   1:  PR[GP1:91,1] = PR[GP1:90,1] + -14.975;
   1:  PR[GP1:91,2] = PR[GP1:90,2] + 38.981;
   1:L PR[91] R[100]mm/sec CNT100;
   1:  PR[GP1:91,1] = PR[GP1:90,1] + -26.046;
   1:  PR[GP1:91,2] = PR[GP1:90,2] + 38.779;
   1:L PR[91] R[100]mm/sec CNT100;
   1:  PR[GP1:91,1] = PR[GP1:90,1] + -28.313;
   1:  PR[GP1:91,2] = PR[GP1:90,2] + 38.036;
   1:L PR[91] R[100]mm/sec CNT100;
   1:  PR[GP1:91,1] = PR[GP1:90,1] + -39.636;
   1:  PR[GP1:91,2] = PR[GP1:90,2] + 33.857;
   1:L PR[91] R[100]mm/sec CNT100;
   1:  PR[GP1:91,1] = PR[GP1:90,1] + -40.541;
   1:  PR[GP1:91,2] = PR[GP1:90,2] + 33.140;
   1:L PR[91] R[100]mm/sec CNT100;
   1:  PR[GP1:91,1] = PR[GP1:90,1] + -50.506;
   1:  PR[GP1:91,2] = PR[GP1:90,2] + 24.916;
   1:L PR[91] R[100]mm/sec CNT100;
   1:  PR[GP1:91,1] = PR[GP1:90,1] + -52.333;
   1:  PR[GP1:91,2] = PR[GP1:90,2] + 21.827;
   1:L PR[91] R[100]mm/sec CNT100;
   1:  PR[GP1:91,1] = PR[GP1:90,1] + -57.539;
   1:  PR[GP1:91,2] = PR[GP1:90,2] + 13.132;
   1:L PR[91] R[100]mm/sec CNT100;
   1:  PR[GP1:91,1] = PR[GP1:90,1] + -57.566;
   1:  PR[GP1:91,2] = PR[GP1:90,2] + 13.038;
   1:L PR[91] R[100]mm/sec CNT100;
   1:  PR[GP1:91,1] = PR[GP1:90,1] + -57.585;
   1:  PR[GP1:91,2] = PR[GP1:90,2] + 12.836;
   1:L PR[91] R[100]mm/sec CNT100;
   1:  PR[GP1:91,1] = PR[GP1:90,1] + -59.969;
   1:  PR[GP1:91,2] = PR[GP1:90,2] + -0.100;
   1:L PR[91] R[100]mm/sec CNT100;
   1:  PR[GP1:91,1] = PR[GP1:90,1] + -59.943;
   1:  PR[GP1:91,2] = PR[GP1:90,2] + -0.390;
   1:L PR[91] R[100]mm/sec CNT100;
   1:  PR[GP1:91,1] = PR[GP1:90,1] + -57.573;
   1:  PR[GP1:91,2] = PR[GP1:90,2] + -13.159;
   1:L PR[91] R[100]mm/sec CNT100;
   1:  PR[GP1:91,1] = PR[GP1:90,1] + -57.531;
   1:  PR[GP1:91,2] = PR[GP1:90,2] + -13.299;
   1:L PR[91] R[100]mm/sec CNT100;
   1:  PR[GP1:91,1] = PR[GP1:90,1] + -57.460;
   1:  PR[GP1:91,2] = PR[GP1:90,2] + -13.440;
   1:L PR[91] R[100]mm/sec CNT100;
   1:  PR[GP1:91,1] = PR[GP1:90,1] + -52.333;
   1:  PR[GP1:91,2] = PR[GP1:90,2] + -21.969;
   1:L PR[91] R[100]mm/sec CNT100;
   1:  PR[GP1:91,1] = PR[GP1:90,1] + -50.500;
   1:  PR[GP1:91,2] = PR[GP1:90,2] + -25.067;
   1:L PR[91] R[100]mm/sec CNT100;
   1:  PR[GP1:91,1] = PR[GP1:90,1] + -40.531;
   1:  PR[GP1:91,2] = PR[GP1:90,2] + -33.290;
   1:L PR[91] R[100]mm/sec CNT100;
   1:  PR[GP1:91,1] = PR[GP1:90,1] + -39.625;
   1:  PR[GP1:91,2] = PR[GP1:90,2] + -34.007;
   1:L PR[91] R[100]mm/sec CNT100;
   1:  PR[GP1:91,1] = PR[GP1:90,1] + -28.299;
   1:  PR[GP1:91,2] = PR[GP1:90,2] + -38.182;
   1:L PR[91] R[100]mm/sec CNT100;
   1:  PR[GP1:91,1] = PR[GP1:90,1] + -26.031;
   1:  PR[GP1:91,2] = PR[GP1:90,2] + -38.926;
   1:L PR[91] R[100]mm/sec CNT100;
   1:  PR[GP1:91,1] = PR[GP1:90,1] + -14.960;
   1:  PR[GP1:91,2] = PR[GP1:90,2] + -39.122;
   1:L PR[91] R[100]mm/sec CNT100;
   1:  PR[GP1:91,1] = PR[GP1:90,1] + -11.340;
   1:  PR[GP1:91,2] = PR[GP1:90,2] + -38.993;
   1:L PR[91] R[100]mm/sec CNT100;
   1:  PR[GP1:91,1] = PR[GP1:90,1] + -1.863;
   1:  PR[GP1:91,2] = PR[GP1:90,2] + -36.043;
   1:L PR[91] R[100]mm/sec CNT100;
   1:  PR[GP1:91,1] = PR[GP1:90,1] + 2.073;
   1:  PR[GP1:91,2] = PR[GP1:90,2] + -36.042;
   1:L PR[91] R[100]mm/sec CNT100;
   1:  PR[GP1:91,1] = PR[GP1:90,1] + 11.551;
   1:  PR[GP1:91,2] = PR[GP1:90,2] + -38.993;
   1:L PR[91] R[100]mm/sec CNT100;
   1:  PR[GP1:91,1] = PR[GP1:90,1] + 15.171;
   1:  PR[GP1:91,2] = PR[GP1:90,2] + -39.122;
   1:L PR[91] R[100]mm/sec CNT100;
   1:  PR[GP1:91,1] = PR[GP1:90,1] + 26.243;
   1:  PR[GP1:91,2] = PR[GP1:90,2] + -38.926;
   1:L PR[91] R[100]mm/sec CNT100;
   1:  PR[GP1:91,1] = PR[GP1:90,1] + 28.510;
   1:  PR[GP1:91,2] = PR[GP1:90,2] + -38.182;
   1:L PR[91] R[100]mm/sec CNT100;
   1:  PR[GP1:91,1] = PR[GP1:90,1] + 39.837;
   1:  PR[GP1:91,2] = PR[GP1:90,2] + -34.010;
   1:L PR[91] R[100]mm/sec CNT100;
   1:  PR[GP1:91,1] = PR[GP1:90,1] + 40.743;
   1:  PR[GP1:91,2] = PR[GP1:90,2] + -33.293;
   1:L PR[91] R[100]mm/sec CNT100;
   1:  PR[GP1:91,1] = PR[GP1:90,1] + 50.715;
   1:  PR[GP1:91,2] = PR[GP1:90,2] + -25.059;
   1:L PR[91] R[100]mm/sec CNT100;
   1:  PR[GP1:91,1] = PR[GP1:90,1] + 50.759;
   1:  PR[GP1:91,2] = PR[GP1:90,2] + -24.985;
   1:L PR[91] R[100]mm/sec CNT100;
   1:  PR[GP1:91,1] = PR[GP1:90,1] + 52.546;
   1:  PR[GP1:91,2] = PR[GP1:90,2] + -21.970;
   1:L PR[91] R[100]mm/sec CNT100;
   1:  PR[GP1:91,1] = PR[GP1:90,1] + 57.750;
   1:  PR[GP1:91,2] = PR[GP1:90,2] + -13.299;
   1:L PR[91] R[100]mm/sec CNT100;
   1:  PR[GP1:91,1] = PR[GP1:90,1] + 57.777;
   1:  PR[GP1:91,2] = PR[GP1:90,2] + -13.208;
   1:L PR[91] R[100]mm/sec CNT100;
   1:  PR[GP1:91,1] = PR[GP1:90,1] + 57.796;
   1:  PR[GP1:91,2] = PR[GP1:90,2] + -13.001;
   1:L PR[91] R[100]mm/sec CNT100;
   1:  PR[GP1:91,1] = PR[GP1:90,1] + 60.182;
   1:  PR[GP1:91,2] = PR[GP1:90,2] + -0.045;
   1:L PR[91] R[100]mm/sec CNT100;
   1:  PR[GP1:91,1] = PR[GP1:90,1] + 60.155;
   1:  PR[GP1:91,2] = PR[GP1:90,2] + 0.256;
   1:L PR[91] R[100]mm/sec CNT100;
   1:  PR[GP1:91,1] = PR[GP1:90,1] + 57.786;
   1:  PR[GP1:91,2] = PR[GP1:90,2] + 13.034;
   1:L PR[91] R[100]mm/sec CNT100;
   1:  PR[GP1:91,1] = PR[GP1:90,1] + 57.746;
   1:  PR[GP1:91,2] = PR[GP1:90,2] + 13.170;
   1:L PR[91] R[100]mm/sec CNT100;
   1:  PR[GP1:91,1] = PR[GP1:90,1] + 57.674;
   1:  PR[GP1:91,2] = PR[GP1:90,2] + 13.309;
   1:L PR[91] R[100]mm/sec CNT100;
   1:  PR[GP1:91,1] = PR[GP1:90,1] + 52.546;
   1:  PR[GP1:91,2] = PR[GP1:90,2] + 21.827;
   1:L PR[91] R[100]mm/sec CNT100;
   1:  PR[GP1:91,1] = PR[GP1:90,1] + 50.718;
   1:  PR[GP1:91,2] = PR[GP1:90,2] + 24.910;
   1:L PR[91] R[100]mm/sec CNT100;
   1:  PR[GP1:91,1] = PR[GP1:90,1] + 40.752;
   1:  PR[GP1:91,2] = PR[GP1:90,2] + 33.144;
   1:L PR[91] R[100]mm/sec CNT100;
   1:  PR[GP1:91,1] = PR[GP1:90,1] + 39.848;
   1:  PR[GP1:91,2] = PR[GP1:90,2] + 33.860;
   1:L PR[91] R[100]mm/sec CNT100;
   1:  PR[GP1:91,1] = PR[GP1:90,1] + 28.524;
   1:  PR[GP1:91,2] = PR[GP1:90,2] + 38.036;
   1:L PR[91] R[100]mm/sec CNT100;
   1:  PR[GP1:91,1] = PR[GP1:90,1] + 26.257;
   1:  PR[GP1:91,2] = PR[GP1:90,2] + 38.780;
   1:L PR[91] R[100]mm/sec CNT100;
   1:  PR[GP1:91,1] = PR[GP1:90,1] + 15.186;
   1:  PR[GP1:91,2] = PR[GP1:90,2] + 38.980;
   1:L PR[91] R[100]mm/sec CNT100;
   1:  PR[GP1:91,1] = PR[GP1:90,1] + 11.565;
   1:  PR[GP1:91,2] = PR[GP1:90,2] + 38.851;
   1:L PR[91] R[100]mm/sec CNT100;
   1:  PR[GP1:91,1] = PR[GP1:90,1] + 2.071;
   1:  PR[GP1:91,2] = PR[GP1:90,2] + 35.917;
   1:L PR[91] R[100]mm/sec CNT100;
   1:  ! -- Layer/Ebene 129 -- !;
   1:  PR[91] = PR[90];
   1:  PR[GP1:91,1] = PR[GP1:90,1] + -1.835;
   1:  PR[GP1:91,2] = PR[GP1:90,2] + 36.091;
   1:  PR[GP1:91,3] = PR[GP1:90,3] + 78.995;
   1:L PR[91] R[100]mm/sec CNT100;
   1:  PR[GP1:91,1] = PR[GP1:90,1] + -11.057;
   1:  PR[GP1:91,2] = PR[GP1:90,2] + 38.940;
   1:L PR[91] R[100]mm/sec CNT100;
   1:  PR[GP1:91,1] = PR[GP1:90,1] + -15.013;
   1:  PR[GP1:91,2] = PR[GP1:90,2] + 39.082;
   1:L PR[91] R[100]mm/sec CNT100;
   1:  PR[GP1:91,1] = PR[GP1:90,1] + -25.784;
   1:  PR[GP1:91,2] = PR[GP1:90,2] + 38.885;
   1:L PR[91] R[100]mm/sec CNT100;
   1:  PR[GP1:91,1] = PR[GP1:90,1] + -28.381;
   1:  PR[GP1:91,2] = PR[GP1:90,2] + 38.034;
   1:L PR[91] R[100]mm/sec CNT100;
   1:  PR[GP1:91,1] = PR[GP1:90,1] + -39.414;
   1:  PR[GP1:91,2] = PR[GP1:90,2] + 33.962;
   1:L PR[91] R[100]mm/sec CNT100;
   1:  PR[GP1:91,1] = PR[GP1:90,1] + -40.601;
   1:  PR[GP1:91,2] = PR[GP1:90,2] + 33.023;
   1:L PR[91] R[100]mm/sec CNT100;
   1:  PR[GP1:91,1] = PR[GP1:90,1] + -50.321;
   1:  PR[GP1:91,2] = PR[GP1:90,2] + 25.000;
   1:L PR[91] R[100]mm/sec CNT100;
   1:  PR[GP1:91,1] = PR[GP1:90,1] + -55.806;
   1:  PR[GP1:91,2] = PR[GP1:90,2] + 15.729;
   1:L PR[91] R[100]mm/sec CNT100;
   1:  PR[GP1:91,1] = PR[GP1:90,1] + -57.336;
   1:  PR[GP1:91,2] = PR[GP1:90,2] + 13.173;
   1:L PR[91] R[100]mm/sec CNT100;
   1:  PR[GP1:91,1] = PR[GP1:90,1] + -57.342;
   1:  PR[GP1:91,2] = PR[GP1:90,2] + 13.142;
   1:L PR[91] R[100]mm/sec CNT100;
   1:  PR[GP1:91,1] = PR[GP1:90,1] + -59.783;
   1:  PR[GP1:91,2] = PR[GP1:90,2] + -0.100;
   1:L PR[91] R[100]mm/sec CNT100;
   1:  PR[GP1:91,1] = PR[GP1:90,1] + -59.771;
   1:  PR[GP1:91,2] = PR[GP1:90,2] + -0.233;
   1:L PR[91] R[100]mm/sec CNT100;
   1:  PR[GP1:91,1] = PR[GP1:90,1] + -57.334;
   1:  PR[GP1:91,2] = PR[GP1:90,2] + -13.322;
   1:L PR[91] R[100]mm/sec CNT100;
   1:  PR[GP1:91,1] = PR[GP1:90,1] + -55.806;
   1:  PR[GP1:91,2] = PR[GP1:90,2] + -15.873;
   1:L PR[91] R[100]mm/sec CNT100;
   1:  PR[GP1:91,1] = PR[GP1:90,1] + -50.315;
   1:  PR[GP1:91,2] = PR[GP1:90,2] + -25.151;
   1:L PR[91] R[100]mm/sec CNT100;
   1:  PR[GP1:91,1] = PR[GP1:90,1] + -40.591;
   1:  PR[GP1:91,2] = PR[GP1:90,2] + -33.172;
   1:L PR[91] R[100]mm/sec CNT100;
   1:  PR[GP1:91,1] = PR[GP1:90,1] + -39.404;
   1:  PR[GP1:91,2] = PR[GP1:90,2] + -34.112;
   1:L PR[91] R[100]mm/sec CNT100;
   1:  PR[GP1:91,1] = PR[GP1:90,1] + -28.368;
   1:  PR[GP1:91,2] = PR[GP1:90,2] + -38.180;
   1:L PR[91] R[100]mm/sec CNT100;
   1:  PR[GP1:91,1] = PR[GP1:90,1] + -25.770;
   1:  PR[GP1:91,2] = PR[GP1:90,2] + -39.032;
   1:L PR[91] R[100]mm/sec CNT100;
   1:  PR[GP1:91,1] = PR[GP1:90,1] + -14.999;
   1:  PR[GP1:91,2] = PR[GP1:90,2] + -39.223;
   1:L PR[91] R[100]mm/sec CNT100;
   1:  PR[GP1:91,1] = PR[GP1:90,1] + -11.043;
   1:  PR[GP1:91,2] = PR[GP1:90,2] + -39.082;
   1:L PR[91] R[100]mm/sec CNT100;
   1:  PR[GP1:91,1] = PR[GP1:90,1] + -1.838;
   1:  PR[GP1:91,2] = PR[GP1:90,2] + -36.217;
   1:L PR[91] R[100]mm/sec CNT100;
   1:  PR[GP1:91,1] = PR[GP1:90,1] + 2.048;
   1:  PR[GP1:91,2] = PR[GP1:90,2] + -36.216;
   1:L PR[91] R[100]mm/sec CNT100;
   1:  PR[GP1:91,1] = PR[GP1:90,1] + 11.254;
   1:  PR[GP1:91,2] = PR[GP1:90,2] + -39.081;
   1:L PR[91] R[100]mm/sec CNT100;
   1:  PR[GP1:91,1] = PR[GP1:90,1] + 15.210;
   1:  PR[GP1:91,2] = PR[GP1:90,2] + -39.222;
   1:L PR[91] R[100]mm/sec CNT100;
   1:  PR[GP1:91,1] = PR[GP1:90,1] + 25.982;
   1:  PR[GP1:91,2] = PR[GP1:90,2] + -39.032;
   1:L PR[91] R[100]mm/sec CNT100;
   1:  PR[GP1:91,1] = PR[GP1:90,1] + 28.579;
   1:  PR[GP1:91,2] = PR[GP1:90,2] + -38.180;
   1:L PR[91] R[100]mm/sec CNT100;
   1:  PR[GP1:91,1] = PR[GP1:90,1] + 39.616;
   1:  PR[GP1:91,2] = PR[GP1:90,2] + -34.115;
   1:L PR[91] R[100]mm/sec CNT100;
   1:  PR[GP1:91,1] = PR[GP1:90,1] + 40.803;
   1:  PR[GP1:91,2] = PR[GP1:90,2] + -33.175;
   1:L PR[91] R[100]mm/sec CNT100;
   1:  PR[GP1:91,1] = PR[GP1:90,1] + 50.530;
   1:  PR[GP1:91,2] = PR[GP1:90,2] + -25.143;
   1:L PR[91] R[100]mm/sec CNT100;
   1:  PR[GP1:91,1] = PR[GP1:90,1] + 50.766;
   1:  PR[GP1:91,2] = PR[GP1:90,2] + -24.753;
   1:L PR[91] R[100]mm/sec CNT100;
   1:  PR[GP1:91,1] = PR[GP1:90,1] + 56.019;
   1:  PR[GP1:91,2] = PR[GP1:90,2] + -15.886;
   1:L PR[91] R[100]mm/sec CNT100;
   1:  PR[GP1:91,1] = PR[GP1:90,1] + 57.546;
   1:  PR[GP1:91,2] = PR[GP1:90,2] + -13.341;
   1:L PR[91] R[100]mm/sec CNT100;
   1:  PR[GP1:91,1] = PR[GP1:90,1] + 59.996;
   1:  PR[GP1:91,2] = PR[GP1:90,2] + -0.045;
   1:L PR[91] R[100]mm/sec CNT100;
   1:  PR[GP1:91,1] = PR[GP1:90,1] + 59.983;
   1:  PR[GP1:91,2] = PR[GP1:90,2] + 0.095;
   1:L PR[91] R[100]mm/sec CNT100;
   1:  PR[GP1:91,1] = PR[GP1:90,1] + 57.548;
   1:  PR[GP1:91,2] = PR[GP1:90,2] + 13.193;
   1:L PR[91] R[100]mm/sec CNT100;
   1:  PR[GP1:91,1] = PR[GP1:90,1] + 56.019;
   1:  PR[GP1:91,2] = PR[GP1:90,2] + 15.742;
   1:L PR[91] R[100]mm/sec CNT100;
   1:  PR[GP1:91,1] = PR[GP1:90,1] + 50.533;
   1:  PR[GP1:91,2] = PR[GP1:90,2] + 24.994;
   1:L PR[91] R[100]mm/sec CNT100;
   1:  PR[GP1:91,1] = PR[GP1:90,1] + 40.812;
   1:  PR[GP1:91,2] = PR[GP1:90,2] + 33.026;
   1:L PR[91] R[100]mm/sec CNT100;
   1:  PR[GP1:91,1] = PR[GP1:90,1] + 39.626;
   1:  PR[GP1:91,2] = PR[GP1:90,2] + 33.965;
   1:L PR[91] R[100]mm/sec CNT100;
   1:  PR[GP1:91,1] = PR[GP1:90,1] + 28.592;
   1:  PR[GP1:91,2] = PR[GP1:90,2] + 38.034;
   1:L PR[91] R[100]mm/sec CNT100;
   1:  PR[GP1:91,1] = PR[GP1:90,1] + 25.995;
   1:  PR[GP1:91,2] = PR[GP1:90,2] + 38.886;
   1:L PR[91] R[100]mm/sec CNT100;
   1:  PR[GP1:91,1] = PR[GP1:90,1] + 15.224;
   1:  PR[GP1:91,2] = PR[GP1:90,2] + 39.081;
   1:L PR[91] R[100]mm/sec CNT100;
   1:  PR[GP1:91,1] = PR[GP1:90,1] + 11.268;
   1:  PR[GP1:91,2] = PR[GP1:90,2] + 38.939;
   1:L PR[91] R[100]mm/sec CNT100;
   1:  PR[GP1:91,1] = PR[GP1:90,1] + 2.046;
   1:  PR[GP1:91,2] = PR[GP1:90,2] + 36.090;
   1:L PR[91] R[100]mm/sec CNT100;
   1:  ! -- Layer/Ebene 130 -- !;
   1:  PR[91] = PR[90];
   1:  PR[GP1:91,1] = PR[GP1:90,1] + -1.810;
   1:  PR[GP1:91,2] = PR[GP1:90,2] + 36.264;
   1:  PR[GP1:91,3] = PR[GP1:90,3] + 79.605;
   1:L PR[91] R[100]mm/sec CNT100;
   1:  PR[GP1:91,1] = PR[GP1:90,1] + -10.759;
   1:  PR[GP1:91,2] = PR[GP1:90,2] + 39.029;
   1:L PR[91] R[100]mm/sec CNT100;
   1:  PR[GP1:91,1] = PR[GP1:90,1] + -15.051;
   1:  PR[GP1:91,2] = PR[GP1:90,2] + 39.183;
   1:L PR[91] R[100]mm/sec CNT100;
   1:  PR[GP1:91,1] = PR[GP1:90,1] + -25.523;
   1:  PR[GP1:91,2] = PR[GP1:90,2] + 38.991;
   1:L PR[91] R[100]mm/sec CNT100;
   1:  PR[GP1:91,1] = PR[GP1:90,1] + -28.449;
   1:  PR[GP1:91,2] = PR[GP1:90,2] + 38.032;
   1:L PR[91] R[100]mm/sec CNT100;
   1:  PR[GP1:91,1] = PR[GP1:90,1] + -39.193;
   1:  PR[GP1:91,2] = PR[GP1:90,2] + 34.067;
   1:L PR[91] R[100]mm/sec CNT100;
   1:  PR[GP1:91,1] = PR[GP1:90,1] + -40.661;
   1:  PR[GP1:91,2] = PR[GP1:90,2] + 32.905;
   1:L PR[91] R[100]mm/sec CNT100;
   1:  PR[GP1:91,1] = PR[GP1:90,1] + -50.136;
   1:  PR[GP1:91,2] = PR[GP1:90,2] + 25.084;
   1:L PR[91] R[100]mm/sec CNT100;
   1:  PR[GP1:91,1] = PR[GP1:90,1] + -57.164;
   1:  PR[GP1:91,2] = PR[GP1:90,2] + 13.211;
   1:L PR[91] R[100]mm/sec CNT100;
   1:  PR[GP1:91,1] = PR[GP1:90,1] + -58.384;
   1:  PR[GP1:91,2] = PR[GP1:90,2] + 6.480;
   1:L PR[91] R[100]mm/sec CNT100;
   1:  PR[GP1:91,1] = PR[GP1:90,1] + -59.592;
   1:  PR[GP1:91,2] = PR[GP1:90,2] + -0.072;
   1:L PR[91] R[100]mm/sec CNT100;
   1:  PR[GP1:91,1] = PR[GP1:90,1] + -58.384;
   1:  PR[GP1:91,2] = PR[GP1:90,2] + -6.623;
   1:L PR[91] R[100]mm/sec CNT100;
   1:  PR[GP1:91,1] = PR[GP1:90,1] + -57.162;
   1:  PR[GP1:91,2] = PR[GP1:90,2] + -13.359;
   1:L PR[91] R[100]mm/sec CNT100;
   1:  PR[GP1:91,1] = PR[GP1:90,1] + -50.131;
   1:  PR[GP1:91,2] = PR[GP1:90,2] + -25.235;
   1:L PR[91] R[100]mm/sec CNT100;
   1:  PR[GP1:91,1] = PR[GP1:90,1] + -40.651;
   1:  PR[GP1:91,2] = PR[GP1:90,2] + -33.054;
   1:L PR[91] R[100]mm/sec CNT100;
   1:  PR[GP1:91,1] = PR[GP1:90,1] + -39.183;
   1:  PR[GP1:91,2] = PR[GP1:90,2] + -34.216;
   1:L PR[91] R[100]mm/sec CNT100;
   1:  PR[GP1:91,1] = PR[GP1:90,1] + -28.437;
   1:  PR[GP1:91,2] = PR[GP1:90,2] + -38.178;
   1:L PR[91] R[100]mm/sec CNT100;
   1:  PR[GP1:91,1] = PR[GP1:90,1] + -25.509;
   1:  PR[GP1:91,2] = PR[GP1:90,2] + -39.138;
   1:L PR[91] R[100]mm/sec CNT100;
   1:  PR[GP1:91,1] = PR[GP1:90,1] + -15.037;
   1:  PR[GP1:91,2] = PR[GP1:90,2] + -39.324;
   1:L PR[91] R[100]mm/sec CNT100;
   1:  PR[GP1:91,1] = PR[GP1:90,1] + -10.746;
   1:  PR[GP1:91,2] = PR[GP1:90,2] + -39.171;
   1:L PR[91] R[100]mm/sec CNT100;
   1:  PR[GP1:91,1] = PR[GP1:90,1] + -1.812;
   1:  PR[GP1:91,2] = PR[GP1:90,2] + -36.391;
   1:L PR[91] R[100]mm/sec CNT100;
   1:  PR[GP1:91,1] = PR[GP1:90,1] + 2.023;
   1:  PR[GP1:91,2] = PR[GP1:90,2] + -36.389;
   1:L PR[91] R[100]mm/sec CNT100;
   1:  PR[GP1:91,1] = PR[GP1:90,1] + 10.958;
   1:  PR[GP1:91,2] = PR[GP1:90,2] + -39.170;
   1:L PR[91] R[100]mm/sec CNT100;
   1:  PR[GP1:91,1] = PR[GP1:90,1] + 15.249;
   1:  PR[GP1:91,2] = PR[GP1:90,2] + -39.323;
   1:L PR[91] R[100]mm/sec CNT100;
   1:  PR[GP1:91,1] = PR[GP1:90,1] + 25.721;
   1:  PR[GP1:91,2] = PR[GP1:90,2] + -39.138;
   1:L PR[91] R[100]mm/sec CNT100;
   1:  PR[GP1:91,1] = PR[GP1:90,1] + 28.648;
   1:  PR[GP1:91,2] = PR[GP1:90,2] + -38.178;
   1:L PR[91] R[100]mm/sec CNT100;
   1:  PR[GP1:91,1] = PR[GP1:90,1] + 39.395;
   1:  PR[GP1:91,2] = PR[GP1:90,2] + -34.219;
   1:L PR[91] R[100]mm/sec CNT100;
   1:  PR[GP1:91,1] = PR[GP1:90,1] + 40.863;
   1:  PR[GP1:91,2] = PR[GP1:90,2] + -33.057;
   1:L PR[91] R[100]mm/sec CNT100;
   1:  PR[GP1:91,1] = PR[GP1:90,1] + 50.346;
   1:  PR[GP1:91,2] = PR[GP1:90,2] + -25.227;
   1:L PR[91] R[100]mm/sec CNT100;
   1:  PR[GP1:91,1] = PR[GP1:90,1] + 50.773;
   1:  PR[GP1:91,2] = PR[GP1:90,2] + -24.520;
   1:L PR[91] R[100]mm/sec CNT100;
   1:  PR[GP1:91,1] = PR[GP1:90,1] + 57.375;
   1:  PR[GP1:91,2] = PR[GP1:90,2] + -13.377;
   1:L PR[91] R[100]mm/sec CNT100;
   1:  PR[GP1:91,1] = PR[GP1:90,1] + 58.596;
   1:  PR[GP1:91,2] = PR[GP1:90,2] + -6.634;
   1:L PR[91] R[100]mm/sec CNT100;
   1:  PR[GP1:91,1] = PR[GP1:90,1] + 59.805;
   1:  PR[GP1:91,2] = PR[GP1:90,2] + -0.072;
   1:L PR[91] R[100]mm/sec CNT100;
   1:  PR[GP1:91,1] = PR[GP1:90,1] + 58.596;
   1:  PR[GP1:91,2] = PR[GP1:90,2] + 6.492;
   1:L PR[91] R[100]mm/sec CNT100;
   1:  PR[GP1:91,1] = PR[GP1:90,1] + 57.377;
   1:  PR[GP1:91,2] = PR[GP1:90,2] + 13.229;
   1:L PR[91] R[100]mm/sec CNT100;
   1:  PR[GP1:91,1] = PR[GP1:90,1] + 50.349;
   1:  PR[GP1:91,2] = PR[GP1:90,2] + 25.079;
   1:L PR[91] R[100]mm/sec CNT100;
   1:  PR[GP1:91,1] = PR[GP1:90,1] + 40.872;
   1:  PR[GP1:91,2] = PR[GP1:90,2] + 32.908;
   1:L PR[91] R[100]mm/sec CNT100;
   1:  PR[GP1:91,1] = PR[GP1:90,1] + 39.405;
   1:  PR[GP1:91,2] = PR[GP1:90,2] + 34.070;
   1:L PR[91] R[100]mm/sec CNT100;
   1:  PR[GP1:91,1] = PR[GP1:90,1] + 28.661;
   1:  PR[GP1:91,2] = PR[GP1:90,2] + 38.032;
   1:L PR[91] R[100]mm/sec CNT100;
   1:  PR[GP1:91,1] = PR[GP1:90,1] + 25.734;
   1:  PR[GP1:91,2] = PR[GP1:90,2] + 38.992;
   1:L PR[91] R[100]mm/sec CNT100;
   1:  PR[GP1:91,1] = PR[GP1:90,1] + 15.263;
   1:  PR[GP1:91,2] = PR[GP1:90,2] + 39.182;
   1:L PR[91] R[100]mm/sec CNT100;
   1:  PR[GP1:91,1] = PR[GP1:90,1] + 10.970;
   1:  PR[GP1:91,2] = PR[GP1:90,2] + 39.028;
   1:L PR[91] R[100]mm/sec CNT100;
   1:  PR[GP1:91,1] = PR[GP1:90,1] + 2.021;
   1:  PR[GP1:91,2] = PR[GP1:90,2] + 36.263;
   1:L PR[91] R[100]mm/sec CNT100;
   1:  ! -- Layer/Ebene 131 -- !;
   1:  PR[91] = PR[90];
   1:  PR[GP1:91,1] = PR[GP1:90,1] + -1.785;
   1:  PR[GP1:91,2] = PR[GP1:90,2] + 36.437;
   1:  PR[GP1:91,3] = PR[GP1:90,3] + 80.215;
   1:L PR[91] R[100]mm/sec CNT100;
   1:  PR[GP1:91,1] = PR[GP1:90,1] + -10.462;
   1:  PR[GP1:91,2] = PR[GP1:90,2] + 39.117;
   1:L PR[91] R[100]mm/sec CNT100;
   1:  PR[GP1:91,1] = PR[GP1:90,1] + -15.089;
   1:  PR[GP1:91,2] = PR[GP1:90,2] + 39.283;
   1:L PR[91] R[100]mm/sec CNT100;
   1:  PR[GP1:91,1] = PR[GP1:90,1] + -25.262;
   1:  PR[GP1:91,2] = PR[GP1:90,2] + 39.098;
   1:L PR[91] R[100]mm/sec CNT100;
   1:  PR[GP1:91,1] = PR[GP1:90,1] + -28.518;
   1:  PR[GP1:91,2] = PR[GP1:90,2] + 38.030;
   1:L PR[91] R[100]mm/sec CNT100;
   1:  PR[GP1:91,1] = PR[GP1:90,1] + -38.971;
   1:  PR[GP1:91,2] = PR[GP1:90,2] + 34.172;
   1:L PR[91] R[100]mm/sec CNT100;
   1:  PR[GP1:91,1] = PR[GP1:90,1] + -40.721;
   1:  PR[GP1:91,2] = PR[GP1:90,2] + 32.787;
   1:L PR[91] R[100]mm/sec CNT100;
   1:  PR[GP1:91,1] = PR[GP1:90,1] + -49.954;
   1:  PR[GP1:91,2] = PR[GP1:90,2] + 25.167;
   1:L PR[91] R[100]mm/sec CNT100;
   1:  PR[GP1:91,1] = PR[GP1:90,1] + -50.573;
   1:  PR[GP1:91,2] = PR[GP1:90,2] + 24.143;
   1:L PR[91] R[100]mm/sec CNT100;
   1:  PR[GP1:91,1] = PR[GP1:90,1] + -57.005;
   1:  PR[GP1:91,2] = PR[GP1:90,2] + 13.258;
   1:L PR[91] R[100]mm/sec CNT100;
   1:  PR[GP1:91,1] = PR[GP1:90,1] + -59.418;
   1:  PR[GP1:91,2] = PR[GP1:90,2] + -0.072;
   1:L PR[91] R[100]mm/sec CNT100;
   1:  PR[GP1:91,1] = PR[GP1:90,1] + -57.155;
   1:  PR[GP1:91,2] = PR[GP1:90,2] + -12.509;
   1:L PR[91] R[100]mm/sec CNT100;
   1:  PR[GP1:91,1] = PR[GP1:90,1] + -57.091;
   1:  PR[GP1:91,2] = PR[GP1:90,2] + -12.935;
   1:L PR[91] R[100]mm/sec CNT100;
   1:  PR[GP1:91,1] = PR[GP1:90,1] + -57.004;
   1:  PR[GP1:91,2] = PR[GP1:90,2] + -13.405;
   1:L PR[91] R[100]mm/sec CNT100;
   1:  PR[GP1:91,1] = PR[GP1:90,1] + -50.568;
   1:  PR[GP1:91,2] = PR[GP1:90,2] + -24.293;
   1:L PR[91] R[100]mm/sec CNT100;
   1:  PR[GP1:91,1] = PR[GP1:90,1] + -49.949;
   1:  PR[GP1:91,2] = PR[GP1:90,2] + -25.317;
   1:L PR[91] R[100]mm/sec CNT100;
   1:  PR[GP1:91,1] = PR[GP1:90,1] + -40.711;
   1:  PR[GP1:91,2] = PR[GP1:90,2] + -32.937;
   1:L PR[91] R[100]mm/sec CNT100;
   1:  PR[GP1:91,1] = PR[GP1:90,1] + -38.962;
   1:  PR[GP1:91,2] = PR[GP1:90,2] + -34.321;
   1:L PR[91] R[100]mm/sec CNT100;
   1:  PR[GP1:91,1] = PR[GP1:90,1] + -28.506;
   1:  PR[GP1:91,2] = PR[GP1:90,2] + -38.175;
   1:L PR[91] R[100]mm/sec CNT100;
   1:  PR[GP1:91,1] = PR[GP1:90,1] + -25.249;
   1:  PR[GP1:91,2] = PR[GP1:90,2] + -39.244;
   1:L PR[91] R[100]mm/sec CNT100;
   1:  PR[GP1:91,1] = PR[GP1:90,1] + -15.076;
   1:  PR[GP1:91,2] = PR[GP1:90,2] + -39.425;
   1:L PR[91] R[100]mm/sec CNT100;
   1:  PR[GP1:91,1] = PR[GP1:90,1] + -10.449;
   1:  PR[GP1:91,2] = PR[GP1:90,2] + -39.260;
   1:L PR[91] R[100]mm/sec CNT100;
   1:  PR[GP1:91,1] = PR[GP1:90,1] + -1.787;
   1:  PR[GP1:91,2] = PR[GP1:90,2] + -36.564;
   1:L PR[91] R[100]mm/sec CNT100;
   1:  PR[GP1:91,1] = PR[GP1:90,1] + 1.998;
   1:  PR[GP1:91,2] = PR[GP1:90,2] + -36.563;
   1:L PR[91] R[100]mm/sec CNT100;
   1:  PR[GP1:91,1] = PR[GP1:90,1] + 10.661;
   1:  PR[GP1:91,2] = PR[GP1:90,2] + -39.259;
   1:L PR[91] R[100]mm/sec CNT100;
   1:  PR[GP1:91,1] = PR[GP1:90,1] + 15.288;
   1:  PR[GP1:91,2] = PR[GP1:90,2] + -39.424;
   1:L PR[91] R[100]mm/sec CNT100;
   1:  PR[GP1:91,1] = PR[GP1:90,1] + 25.460;
   1:  PR[GP1:91,2] = PR[GP1:90,2] + -39.244;
   1:L PR[91] R[100]mm/sec CNT100;
   1:  PR[GP1:91,1] = PR[GP1:90,1] + 28.717;
   1:  PR[GP1:91,2] = PR[GP1:90,2] + -38.176;
   1:L PR[91] R[100]mm/sec CNT100;
   1:  PR[GP1:91,1] = PR[GP1:90,1] + 39.174;
   1:  PR[GP1:91,2] = PR[GP1:90,2] + -34.324;
   1:L PR[91] R[100]mm/sec CNT100;
   1:  PR[GP1:91,1] = PR[GP1:90,1] + 40.924;
   1:  PR[GP1:91,2] = PR[GP1:90,2] + -32.939;
   1:L PR[91] R[100]mm/sec CNT100;
   1:  PR[GP1:91,1] = PR[GP1:90,1] + 50.161;
   1:  PR[GP1:91,2] = PR[GP1:90,2] + -25.311;
   1:L PR[91] R[100]mm/sec CNT100;
   1:  PR[GP1:91,1] = PR[GP1:90,1] + 50.781;
   1:  PR[GP1:91,2] = PR[GP1:90,2] + -24.287;
   1:L PR[91] R[100]mm/sec CNT100;
   1:  PR[GP1:91,1] = PR[GP1:90,1] + 57.217;
   1:  PR[GP1:91,2] = PR[GP1:90,2] + -13.423;
   1:L PR[91] R[100]mm/sec CNT100;
   1:  PR[GP1:91,1] = PR[GP1:90,1] + 59.632;
   1:  PR[GP1:91,2] = PR[GP1:90,2] + -0.072;
   1:L PR[91] R[100]mm/sec CNT100;
   1:  PR[GP1:91,1] = PR[GP1:90,1] + 57.370;
   1:  PR[GP1:91,2] = PR[GP1:90,2] + 12.373;
   1:L PR[91] R[100]mm/sec CNT100;
   1:  PR[GP1:91,1] = PR[GP1:90,1] + 57.216;
   1:  PR[GP1:91,2] = PR[GP1:90,2] + 13.279;
   1:L PR[91] R[100]mm/sec CNT100;
   1:  PR[GP1:91,1] = PR[GP1:90,1] + 50.786;
   1:  PR[GP1:91,2] = PR[GP1:90,2] + 24.137;
   1:L PR[91] R[100]mm/sec CNT100;
   1:  PR[GP1:91,1] = PR[GP1:90,1] + 50.166;
   1:  PR[GP1:91,2] = PR[GP1:90,2] + 25.161;
   1:L PR[91] R[100]mm/sec CNT100;
   1:  PR[GP1:91,1] = PR[GP1:90,1] + 40.932;
   1:  PR[GP1:91,2] = PR[GP1:90,2] + 32.790;
   1:L PR[91] R[100]mm/sec CNT100;
   1:  PR[GP1:91,1] = PR[GP1:90,1] + 39.183;
   1:  PR[GP1:91,2] = PR[GP1:90,2] + 34.175;
   1:L PR[91] R[100]mm/sec CNT100;
   1:  PR[GP1:91,1] = PR[GP1:90,1] + 28.729;
   1:  PR[GP1:91,2] = PR[GP1:90,2] + 38.030;
   1:L PR[91] R[100]mm/sec CNT100;
   1:  PR[GP1:91,1] = PR[GP1:90,1] + 25.473;
   1:  PR[GP1:91,2] = PR[GP1:90,2] + 39.098;
   1:L PR[91] R[100]mm/sec CNT100;
   1:  PR[GP1:91,1] = PR[GP1:90,1] + 15.301;
   1:  PR[GP1:91,2] = PR[GP1:90,2] + 39.282;
   1:L PR[91] R[100]mm/sec CNT100;
   1:  PR[GP1:91,1] = PR[GP1:90,1] + 10.673;
   1:  PR[GP1:91,2] = PR[GP1:90,2] + 39.117;
   1:L PR[91] R[100]mm/sec CNT100;
   1:  PR[GP1:91,1] = PR[GP1:90,1] + 1.996;
   1:  PR[GP1:91,2] = PR[GP1:90,2] + 36.436;
   1:L PR[91] R[100]mm/sec CNT100;
   1:  ! -- Layer/Ebene 132 -- !;
   1:  PR[91] = PR[90];
   1:  PR[GP1:91,1] = PR[GP1:90,1] + -1.759;
   1:  PR[GP1:91,2] = PR[GP1:90,2] + 36.611;
   1:  PR[GP1:91,3] = PR[GP1:90,3] + 80.825;
   1:L PR[91] R[100]mm/sec CNT100;
   1:  PR[GP1:91,1] = PR[GP1:90,1] + -10.164;
   1:  PR[GP1:91,2] = PR[GP1:90,2] + 39.206;
   1:L PR[91] R[100]mm/sec CNT100;
   1:  PR[GP1:91,1] = PR[GP1:90,1] + -15.128;
   1:  PR[GP1:91,2] = PR[GP1:90,2] + 39.384;
   1:L PR[91] R[100]mm/sec CNT100;
   1:  PR[GP1:91,1] = PR[GP1:90,1] + -25.000;
   1:  PR[GP1:91,2] = PR[GP1:90,2] + 39.204;
   1:L PR[91] R[100]mm/sec CNT100;
   1:  PR[GP1:91,1] = PR[GP1:90,1] + -28.587;
   1:  PR[GP1:91,2] = PR[GP1:90,2] + 38.028;
   1:L PR[91] R[100]mm/sec CNT100;
   1:  PR[GP1:91,1] = PR[GP1:90,1] + -38.750;
   1:  PR[GP1:91,2] = PR[GP1:90,2] + 34.277;
   1:L PR[91] R[100]mm/sec CNT100;
   1:  PR[GP1:91,1] = PR[GP1:90,1] + -40.781;
   1:  PR[GP1:91,2] = PR[GP1:90,2] + 32.670;
   1:L PR[91] R[100]mm/sec CNT100;
   1:  PR[GP1:91,1] = PR[GP1:90,1] + -49.769;
   1:  PR[GP1:91,2] = PR[GP1:90,2] + 25.251;
   1:L PR[91] R[100]mm/sec CNT100;
   1:  PR[GP1:91,1] = PR[GP1:90,1] + -50.580;
   1:  PR[GP1:91,2] = PR[GP1:90,2] + 23.910;
   1:L PR[91] R[100]mm/sec CNT100;
   1:  PR[GP1:91,1] = PR[GP1:90,1] + -56.847;
   1:  PR[GP1:91,2] = PR[GP1:90,2] + 13.305;
   1:L PR[91] R[100]mm/sec CNT100;
   1:  PR[GP1:91,1] = PR[GP1:90,1] + -59.188;
   1:  PR[GP1:91,2] = PR[GP1:90,2] + 0.388;
   1:L PR[91] R[100]mm/sec CNT100;
   1:  PR[GP1:91,1] = PR[GP1:90,1] + -59.262;
   1:  PR[GP1:91,2] = PR[GP1:90,2] + -0.066;
   1:L PR[91] R[100]mm/sec CNT100;
   1:  PR[GP1:91,1] = PR[GP1:90,1] + -57.106;
   1:  PR[GP1:91,2] = PR[GP1:90,2] + -11.910;
   1:L PR[91] R[100]mm/sec CNT100;
   1:  PR[GP1:91,1] = PR[GP1:90,1] + -57.001;
   1:  PR[GP1:91,2] = PR[GP1:90,2] + -12.610;
   1:L PR[91] R[100]mm/sec CNT100;
   1:  PR[GP1:91,1] = PR[GP1:90,1] + -56.846;
   1:  PR[GP1:91,2] = PR[GP1:90,2] + -13.452;
   1:L PR[91] R[100]mm/sec CNT100;
   1:  PR[GP1:91,1] = PR[GP1:90,1] + -50.575;
   1:  PR[GP1:91,2] = PR[GP1:90,2] + -24.060;
   1:L PR[91] R[100]mm/sec CNT100;
   1:  PR[GP1:91,1] = PR[GP1:90,1] + -49.764;
   1:  PR[GP1:91,2] = PR[GP1:90,2] + -25.401;
   1:L PR[91] R[100]mm/sec CNT100;
   1:  PR[GP1:91,1] = PR[GP1:90,1] + -40.771;
   1:  PR[GP1:91,2] = PR[GP1:90,2] + -32.819;
   1:L PR[91] R[100]mm/sec CNT100;
   1:  PR[GP1:91,1] = PR[GP1:90,1] + -38.741;
   1:  PR[GP1:91,2] = PR[GP1:90,2] + -34.426;
   1:L PR[91] R[100]mm/sec CNT100;
   1:  PR[GP1:91,1] = PR[GP1:90,1] + -28.575;
   1:  PR[GP1:91,2] = PR[GP1:90,2] + -38.173;
   1:L PR[91] R[100]mm/sec CNT100;
   1:  PR[GP1:91,1] = PR[GP1:90,1] + -24.988;
   1:  PR[GP1:91,2] = PR[GP1:90,2] + -39.350;
   1:L PR[91] R[100]mm/sec CNT100;
   1:  PR[GP1:91,1] = PR[GP1:90,1] + -15.115;
   1:  PR[GP1:91,2] = PR[GP1:90,2] + -39.525;
   1:L PR[91] R[100]mm/sec CNT100;
   1:  PR[GP1:91,1] = PR[GP1:90,1] + -10.152;
   1:  PR[GP1:91,2] = PR[GP1:90,2] + -39.348;
   1:L PR[91] R[100]mm/sec CNT100;
   1:  PR[GP1:91,1] = PR[GP1:90,1] + -1.762;
   1:  PR[GP1:91,2] = PR[GP1:90,2] + -36.738;
   1:L PR[91] R[100]mm/sec CNT100;
   1:  PR[GP1:91,1] = PR[GP1:90,1] + 1.973;
   1:  PR[GP1:91,2] = PR[GP1:90,2] + -36.737;
   1:L PR[91] R[100]mm/sec CNT100;
   1:  PR[GP1:91,1] = PR[GP1:90,1] + 10.364;
   1:  PR[GP1:91,2] = PR[GP1:90,2] + -39.348;
   1:L PR[91] R[100]mm/sec CNT100;
   1:  PR[GP1:91,1] = PR[GP1:90,1] + 15.326;
   1:  PR[GP1:91,2] = PR[GP1:90,2] + -39.525;
   1:L PR[91] R[100]mm/sec CNT100;
   1:  PR[GP1:91,1] = PR[GP1:90,1] + 25.200;
   1:  PR[GP1:91,2] = PR[GP1:90,2] + -39.351;
   1:L PR[91] R[100]mm/sec CNT100;
   1:  PR[GP1:91,1] = PR[GP1:90,1] + 28.786;
   1:  PR[GP1:91,2] = PR[GP1:90,2] + -38.174;
   1:L PR[91] R[100]mm/sec CNT100;
   1:  PR[GP1:91,1] = PR[GP1:90,1] + 38.953;
   1:  PR[GP1:91,2] = PR[GP1:90,2] + -34.429;
   1:L PR[91] R[100]mm/sec CNT100;
   1:  PR[GP1:91,1] = PR[GP1:90,1] + 40.983;
   1:  PR[GP1:91,2] = PR[GP1:90,2] + -32.821;
   1:L PR[91] R[100]mm/sec CNT100;
   1:  PR[GP1:91,1] = PR[GP1:90,1] + 49.977;
   1:  PR[GP1:91,2] = PR[GP1:90,2] + -25.395;
   1:L PR[91] R[100]mm/sec CNT100;
   1:  PR[GP1:91,1] = PR[GP1:90,1] + 50.788;
   1:  PR[GP1:91,2] = PR[GP1:90,2] + -24.054;
   1:L PR[91] R[100]mm/sec CNT100;
   1:  PR[GP1:91,1] = PR[GP1:90,1] + 57.058;
   1:  PR[GP1:91,2] = PR[GP1:90,2] + -13.470;
   1:L PR[91] R[100]mm/sec CNT100;
   1:  PR[GP1:91,1] = PR[GP1:90,1] + 59.402;
   1:  PR[GP1:91,2] = PR[GP1:90,2] + -0.532;
   1:L PR[91] R[100]mm/sec CNT100;
   1:  PR[GP1:91,1] = PR[GP1:90,1] + 59.475;
   1:  PR[GP1:91,2] = PR[GP1:90,2] + -0.078;
   1:L PR[91] R[100]mm/sec CNT100;
   1:  PR[GP1:91,1] = PR[GP1:90,1] + 57.320;
   1:  PR[GP1:91,2] = PR[GP1:90,2] + 11.779;
   1:L PR[91] R[100]mm/sec CNT100;
   1:  PR[GP1:91,1] = PR[GP1:90,1] + 57.215;
   1:  PR[GP1:91,2] = PR[GP1:90,2] + 12.480;
   1:L PR[91] R[100]mm/sec CNT100;
   1:  PR[GP1:91,1] = PR[GP1:90,1] + 57.060;
   1:  PR[GP1:91,2] = PR[GP1:90,2] + 13.322;
   1:L PR[91] R[100]mm/sec CNT100;
   1:  PR[GP1:91,1] = PR[GP1:90,1] + 50.793;
   1:  PR[GP1:91,2] = PR[GP1:90,2] + 23.905;
   1:L PR[91] R[100]mm/sec CNT100;
   1:  PR[GP1:91,1] = PR[GP1:90,1] + 49.982;
   1:  PR[GP1:91,2] = PR[GP1:90,2] + 25.245;
   1:L PR[91] R[100]mm/sec CNT100;
   1:  PR[GP1:91,1] = PR[GP1:90,1] + 40.992;
   1:  PR[GP1:91,2] = PR[GP1:90,2] + 32.673;
   1:L PR[91] R[100]mm/sec CNT100;
   1:  PR[GP1:91,1] = PR[GP1:90,1] + 38.962;
   1:  PR[GP1:91,2] = PR[GP1:90,2] + 34.280;
   1:L PR[91] R[100]mm/sec CNT100;
   1:  PR[GP1:91,1] = PR[GP1:90,1] + 28.798;
   1:  PR[GP1:91,2] = PR[GP1:90,2] + 38.028;
   1:L PR[91] R[100]mm/sec CNT100;
   1:  PR[GP1:91,1] = PR[GP1:90,1] + 25.212;
   1:  PR[GP1:91,2] = PR[GP1:90,2] + 39.204;
   1:L PR[91] R[100]mm/sec CNT100;
   1:  PR[GP1:91,1] = PR[GP1:90,1] + 15.339;
   1:  PR[GP1:91,2] = PR[GP1:90,2] + 39.383;
   1:L PR[91] R[100]mm/sec CNT100;
   1:  PR[GP1:91,1] = PR[GP1:90,1] + 10.375;
   1:  PR[GP1:91,2] = PR[GP1:90,2] + 39.205;
   1:L PR[91] R[100]mm/sec CNT100;
   1:  PR[GP1:91,1] = PR[GP1:90,1] + 1.971;
   1:  PR[GP1:91,2] = PR[GP1:90,2] + 36.609;
   1:L PR[91] R[100]mm/sec CNT100;
   1:  ! -- Layer/Ebene 133 -- !;
   1:  PR[91] = PR[90];
   1:  PR[GP1:91,1] = PR[GP1:90,1] + -1.734;
   1:  PR[GP1:91,2] = PR[GP1:90,2] + 36.784;
   1:  PR[GP1:91,3] = PR[GP1:90,3] + 81.435;
   1:L PR[91] R[100]mm/sec CNT100;
   1:  PR[GP1:91,1] = PR[GP1:90,1] + -9.866;
   1:  PR[GP1:91,2] = PR[GP1:90,2] + 39.295;
   1:L PR[91] R[100]mm/sec CNT100;
   1:  PR[GP1:91,1] = PR[GP1:90,1] + -15.166;
   1:  PR[GP1:91,2] = PR[GP1:90,2] + 39.485;
   1:L PR[91] R[100]mm/sec CNT100;
   1:  PR[GP1:91,1] = PR[GP1:90,1] + -24.739;
   1:  PR[GP1:91,2] = PR[GP1:90,2] + 39.310;
   1:L PR[91] R[100]mm/sec CNT100;
   1:  PR[GP1:91,1] = PR[GP1:90,1] + -28.655;
   1:  PR[GP1:91,2] = PR[GP1:90,2] + 38.026;
   1:L PR[91] R[100]mm/sec CNT100;
   1:  PR[GP1:91,1] = PR[GP1:90,1] + -38.528;
   1:  PR[GP1:91,2] = PR[GP1:90,2] + 34.382;
   1:L PR[91] R[100]mm/sec CNT100;
   1:  PR[GP1:91,1] = PR[GP1:90,1] + -40.840;
   1:  PR[GP1:91,2] = PR[GP1:90,2] + 32.552;
   1:L PR[91] R[100]mm/sec CNT100;
   1:  PR[GP1:91,1] = PR[GP1:90,1] + -49.584;
   1:  PR[GP1:91,2] = PR[GP1:90,2] + 25.335;
   1:L PR[91] R[100]mm/sec CNT100;
   1:  PR[GP1:91,1] = PR[GP1:90,1] + -50.587;
   1:  PR[GP1:91,2] = PR[GP1:90,2] + 23.677;
   1:L PR[91] R[100]mm/sec CNT100;
   1:  PR[GP1:91,1] = PR[GP1:90,1] + -56.688;
   1:  PR[GP1:91,2] = PR[GP1:90,2] + 13.352;
   1:L PR[91] R[100]mm/sec CNT100;
   1:  PR[GP1:91,1] = PR[GP1:90,1] + -58.968;
   1:  PR[GP1:91,2] = PR[GP1:90,2] + 0.775;
   1:L PR[91] R[100]mm/sec CNT100;
   1:  PR[GP1:91,1] = PR[GP1:90,1] + -59.104;
   1:  PR[GP1:91,2] = PR[GP1:90,2] + -0.066;
   1:L PR[91] R[100]mm/sec CNT100;
   1:  PR[GP1:91,1] = PR[GP1:90,1] + -57.057;
   1:  PR[GP1:91,2] = PR[GP1:90,2] + -11.312;
   1:L PR[91] R[100]mm/sec CNT100;
   1:  PR[GP1:91,1] = PR[GP1:90,1] + -56.911;
   1:  PR[GP1:91,2] = PR[GP1:90,2] + -12.284;
   1:L PR[91] R[100]mm/sec CNT100;
   1:  PR[GP1:91,1] = PR[GP1:90,1] + -56.687;
   1:  PR[GP1:91,2] = PR[GP1:90,2] + -13.499;
   1:L PR[91] R[100]mm/sec CNT100;
   1:  PR[GP1:91,1] = PR[GP1:90,1] + -50.582;
   1:  PR[GP1:91,2] = PR[GP1:90,2] + -23.827;
   1:L PR[91] R[100]mm/sec CNT100;
   1:  PR[GP1:91,1] = PR[GP1:90,1] + -49.580;
   1:  PR[GP1:91,2] = PR[GP1:90,2] + -25.485;
   1:L PR[91] R[100]mm/sec CNT100;
   1:  PR[GP1:91,1] = PR[GP1:90,1] + -40.831;
   1:  PR[GP1:91,2] = PR[GP1:90,2] + -32.701;
   1:L PR[91] R[100]mm/sec CNT100;
   1:  PR[GP1:91,1] = PR[GP1:90,1] + -38.519;
   1:  PR[GP1:91,2] = PR[GP1:90,2] + -34.531;
   1:L PR[91] R[100]mm/sec CNT100;
   1:  PR[GP1:91,1] = PR[GP1:90,1] + -28.643;
   1:  PR[GP1:91,2] = PR[GP1:90,2] + -38.171;
   1:L PR[91] R[100]mm/sec CNT100;
   1:  PR[GP1:91,1] = PR[GP1:90,1] + -24.727;
   1:  PR[GP1:91,2] = PR[GP1:90,2] + -39.456;
   1:L PR[91] R[100]mm/sec CNT100;
   1:  PR[GP1:91,1] = PR[GP1:90,1] + -15.153;
   1:  PR[GP1:91,2] = PR[GP1:90,2] + -39.626;
   1:L PR[91] R[100]mm/sec CNT100;
   1:  PR[GP1:91,1] = PR[GP1:90,1] + -9.855;
   1:  PR[GP1:91,2] = PR[GP1:90,2] + -39.437;
   1:L PR[91] R[100]mm/sec CNT100;
   1:  PR[GP1:91,1] = PR[GP1:90,1] + -1.736;
   1:  PR[GP1:91,2] = PR[GP1:90,2] + -36.912;
   1:L PR[91] R[100]mm/sec CNT100;
   1:  PR[GP1:91,1] = PR[GP1:90,1] + 1.948;
   1:  PR[GP1:91,2] = PR[GP1:90,2] + -36.911;
   1:L PR[91] R[100]mm/sec CNT100;
   1:  PR[GP1:91,1] = PR[GP1:90,1] + 10.067;
   1:  PR[GP1:91,2] = PR[GP1:90,2] + -39.437;
   1:L PR[91] R[100]mm/sec CNT100;
   1:  PR[GP1:91,1] = PR[GP1:90,1] + 15.365;
   1:  PR[GP1:91,2] = PR[GP1:90,2] + -39.625;
   1:L PR[91] R[100]mm/sec CNT100;
   1:  PR[GP1:91,1] = PR[GP1:90,1] + 24.939;
   1:  PR[GP1:91,2] = PR[GP1:90,2] + -39.457;
   1:L PR[91] R[100]mm/sec CNT100;
   1:  PR[GP1:91,1] = PR[GP1:90,1] + 28.855;
   1:  PR[GP1:91,2] = PR[GP1:90,2] + -38.172;
   1:L PR[91] R[100]mm/sec CNT100;
   1:  PR[GP1:91,1] = PR[GP1:90,1] + 38.732;
   1:  PR[GP1:91,2] = PR[GP1:90,2] + -34.534;
   1:L PR[91] R[100]mm/sec CNT100;
   1:  PR[GP1:91,1] = PR[GP1:90,1] + 41.044;
   1:  PR[GP1:91,2] = PR[GP1:90,2] + -32.703;
   1:L PR[91] R[100]mm/sec CNT100;
   1:  PR[GP1:91,1] = PR[GP1:90,1] + 49.792;
   1:  PR[GP1:91,2] = PR[GP1:90,2] + -25.479;
   1:L PR[91] R[100]mm/sec CNT100;
   1:  PR[GP1:91,1] = PR[GP1:90,1] + 50.795;
   1:  PR[GP1:91,2] = PR[GP1:90,2] + -23.821;
   1:L PR[91] R[100]mm/sec CNT100;
   1:  PR[GP1:91,1] = PR[GP1:90,1] + 56.900;
   1:  PR[GP1:91,2] = PR[GP1:90,2] + -13.517;
   1:L PR[91] R[100]mm/sec CNT100;
   1:  PR[GP1:91,1] = PR[GP1:90,1] + 59.181;
   1:  PR[GP1:91,2] = PR[GP1:90,2] + -0.920;
   1:L PR[91] R[100]mm/sec CNT100;
   1:  PR[GP1:91,1] = PR[GP1:90,1] + 59.317;
   1:  PR[GP1:91,2] = PR[GP1:90,2] + -0.078;
   1:L PR[91] R[100]mm/sec CNT100;
   1:  PR[GP1:91,1] = PR[GP1:90,1] + 57.271;
   1:  PR[GP1:91,2] = PR[GP1:90,2] + 11.180;
   1:L PR[91] R[100]mm/sec CNT100;
   1:  PR[GP1:91,1] = PR[GP1:90,1] + 57.126;
   1:  PR[GP1:91,2] = PR[GP1:90,2] + 12.154;
   1:L PR[91] R[100]mm/sec CNT100;
   1:  PR[GP1:91,1] = PR[GP1:90,1] + 56.902;
   1:  PR[GP1:91,2] = PR[GP1:90,2] + 13.369;
   1:L PR[91] R[100]mm/sec CNT100;
   1:  PR[GP1:91,1] = PR[GP1:90,1] + 50.800;
   1:  PR[GP1:91,2] = PR[GP1:90,2] + 23.672;
   1:L PR[91] R[100]mm/sec CNT100;
   1:  PR[GP1:91,1] = PR[GP1:90,1] + 49.797;
   1:  PR[GP1:91,2] = PR[GP1:90,2] + 25.330;
   1:L PR[91] R[100]mm/sec CNT100;
   1:  PR[GP1:91,1] = PR[GP1:90,1] + 41.052;
   1:  PR[GP1:91,2] = PR[GP1:90,2] + 32.555;
   1:L PR[91] R[100]mm/sec CNT100;
   1:  PR[GP1:91,1] = PR[GP1:90,1] + 38.740;
   1:  PR[GP1:91,2] = PR[GP1:90,2] + 34.385;
   1:L PR[91] R[100]mm/sec CNT100;
   1:  PR[GP1:91,1] = PR[GP1:90,1] + 28.866;
   1:  PR[GP1:91,2] = PR[GP1:90,2] + 38.026;
   1:L PR[91] R[100]mm/sec CNT100;
   1:  PR[GP1:91,1] = PR[GP1:90,1] + 24.950;
   1:  PR[GP1:91,2] = PR[GP1:90,2] + 39.310;
   1:L PR[91] R[100]mm/sec CNT100;
   1:  PR[GP1:91,1] = PR[GP1:90,1] + 15.377;
   1:  PR[GP1:91,2] = PR[GP1:90,2] + 39.484;
   1:L PR[91] R[100]mm/sec CNT100;
   1:  PR[GP1:91,1] = PR[GP1:90,1] + 10.078;
   1:  PR[GP1:91,2] = PR[GP1:90,2] + 39.294;
   1:L PR[91] R[100]mm/sec CNT100;
   1:  PR[GP1:91,1] = PR[GP1:90,1] + 1.946;
   1:  PR[GP1:91,2] = PR[GP1:90,2] + 36.783;
   1:L PR[91] R[100]mm/sec CNT100;
   1:  ! -- Layer/Ebene 134 -- !;
   1:  PR[91] = PR[90];
   1:  PR[GP1:91,1] = PR[GP1:90,1] + -1.709;
   1:  PR[GP1:91,2] = PR[GP1:90,2] + 36.957;
   1:  PR[GP1:91,3] = PR[GP1:90,3] + 82.045;
   1:L PR[91] R[100]mm/sec CNT100;
   1:  PR[GP1:91,1] = PR[GP1:90,1] + -9.569;
   1:  PR[GP1:91,2] = PR[GP1:90,2] + 39.383;
   1:L PR[91] R[100]mm/sec CNT100;
   1:  PR[GP1:91,1] = PR[GP1:90,1] + -15.204;
   1:  PR[GP1:91,2] = PR[GP1:90,2] + 39.585;
   1:L PR[91] R[100]mm/sec CNT100;
   1:  PR[GP1:91,1] = PR[GP1:90,1] + -24.477;
   1:  PR[GP1:91,2] = PR[GP1:90,2] + 39.416;
   1:L PR[91] R[100]mm/sec CNT100;
   1:  PR[GP1:91,1] = PR[GP1:90,1] + -28.723;
   1:  PR[GP1:91,2] = PR[GP1:90,2] + 38.024;
   1:L PR[91] R[100]mm/sec CNT100;
   1:  PR[GP1:91,1] = PR[GP1:90,1] + -38.307;
   1:  PR[GP1:91,2] = PR[GP1:90,2] + 34.487;
   1:L PR[91] R[100]mm/sec CNT100;
   1:  PR[GP1:91,1] = PR[GP1:90,1] + -40.900;
   1:  PR[GP1:91,2] = PR[GP1:90,2] + 32.434;
   1:L PR[91] R[100]mm/sec CNT100;
   1:  PR[GP1:91,1] = PR[GP1:90,1] + -49.400;
   1:  PR[GP1:91,2] = PR[GP1:90,2] + 25.419;
   1:L PR[91] R[100]mm/sec CNT100;
   1:  PR[GP1:91,1] = PR[GP1:90,1] + -50.594;
   1:  PR[GP1:91,2] = PR[GP1:90,2] + 23.445;
   1:L PR[91] R[100]mm/sec CNT100;
   1:  PR[GP1:91,1] = PR[GP1:90,1] + -56.530;
   1:  PR[GP1:91,2] = PR[GP1:90,2] + 13.400;
   1:L PR[91] R[100]mm/sec CNT100;
   1:  PR[GP1:91,1] = PR[GP1:90,1] + -58.748;
   1:  PR[GP1:91,2] = PR[GP1:90,2] + 1.164;
   1:L PR[91] R[100]mm/sec CNT100;
   1:  PR[GP1:91,1] = PR[GP1:90,1] + -58.946;
   1:  PR[GP1:91,2] = PR[GP1:90,2] + -0.066;
   1:L PR[91] R[100]mm/sec CNT100;
   1:  PR[GP1:91,1] = PR[GP1:90,1] + -57.008;
   1:  PR[GP1:91,2] = PR[GP1:90,2] + -10.713;
   1:L PR[91] R[100]mm/sec CNT100;
   1:  PR[GP1:91,1] = PR[GP1:90,1] + -56.822;
   1:  PR[GP1:91,2] = PR[GP1:90,2] + -11.959;
   1:L PR[91] R[100]mm/sec CNT100;
   1:  PR[GP1:91,1] = PR[GP1:90,1] + -56.529;
   1:  PR[GP1:91,2] = PR[GP1:90,2] + -13.546;
   1:L PR[91] R[100]mm/sec CNT100;
   1:  PR[GP1:91,1] = PR[GP1:90,1] + -50.589;
   1:  PR[GP1:91,2] = PR[GP1:90,2] + -23.594;
   1:L PR[91] R[100]mm/sec CNT100;
   1:  PR[GP1:91,1] = PR[GP1:90,1] + -49.395;
   1:  PR[GP1:91,2] = PR[GP1:90,2] + -25.569;
   1:L PR[91] R[100]mm/sec CNT100;
   1:  PR[GP1:91,1] = PR[GP1:90,1] + -40.892;
   1:  PR[GP1:91,2] = PR[GP1:90,2] + -32.583;
   1:L PR[91] R[100]mm/sec CNT100;
   1:  PR[GP1:91,1] = PR[GP1:90,1] + -38.298;
   1:  PR[GP1:91,2] = PR[GP1:90,2] + -34.636;
   1:L PR[91] R[100]mm/sec CNT100;
   1:  PR[GP1:91,1] = PR[GP1:90,1] + -28.712;
   1:  PR[GP1:91,2] = PR[GP1:90,2] + -38.169;
   1:L PR[91] R[100]mm/sec CNT100;
   1:  PR[GP1:91,1] = PR[GP1:90,1] + -24.466;
   1:  PR[GP1:91,2] = PR[GP1:90,2] + -39.562;
   1:L PR[91] R[100]mm/sec CNT100;
   1:  PR[GP1:91,1] = PR[GP1:90,1] + -15.192;
   1:  PR[GP1:91,2] = PR[GP1:90,2] + -39.727;
   1:L PR[91] R[100]mm/sec CNT100;
   1:  PR[GP1:91,1] = PR[GP1:90,1] + -9.558;
   1:  PR[GP1:91,2] = PR[GP1:90,2] + -39.526;
   1:L PR[91] R[100]mm/sec CNT100;
   1:  PR[GP1:91,1] = PR[GP1:90,1] + -1.711;
   1:  PR[GP1:91,2] = PR[GP1:90,2] + -37.085;
   1:L PR[91] R[100]mm/sec CNT100;
   1:  PR[GP1:91,1] = PR[GP1:90,1] + 1.923;
   1:  PR[GP1:91,2] = PR[GP1:90,2] + -37.084;
   1:L PR[91] R[100]mm/sec CNT100;
   1:  PR[GP1:91,1] = PR[GP1:90,1] + 9.771;
   1:  PR[GP1:91,2] = PR[GP1:90,2] + -39.525;
   1:L PR[91] R[100]mm/sec CNT100;
   1:  PR[GP1:91,1] = PR[GP1:90,1] + 15.404;
   1:  PR[GP1:91,2] = PR[GP1:90,2] + -39.726;
   1:L PR[91] R[100]mm/sec CNT100;
   1:  PR[GP1:91,1] = PR[GP1:90,1] + 24.678;
   1:  PR[GP1:91,2] = PR[GP1:90,2] + -39.563;
   1:L PR[91] R[100]mm/sec CNT100;
   1:  PR[GP1:91,1] = PR[GP1:90,1] + 28.924;
   1:  PR[GP1:91,2] = PR[GP1:90,2] + -38.170;
   1:L PR[91] R[100]mm/sec CNT100;
   1:  PR[GP1:91,1] = PR[GP1:90,1] + 38.511;
   1:  PR[GP1:91,2] = PR[GP1:90,2] + -34.638;
   1:L PR[91] R[100]mm/sec CNT100;
   1:  PR[GP1:91,1] = PR[GP1:90,1] + 41.104;
   1:  PR[GP1:91,2] = PR[GP1:90,2] + -32.585;
   1:L PR[91] R[100]mm/sec CNT100;
   1:  PR[GP1:91,1] = PR[GP1:90,1] + 49.608;
   1:  PR[GP1:91,2] = PR[GP1:90,2] + -25.563;
   1:L PR[91] R[100]mm/sec CNT100;
   1:  PR[GP1:91,1] = PR[GP1:90,1] + 50.802;
   1:  PR[GP1:91,2] = PR[GP1:90,2] + -23.589;
   1:L PR[91] R[100]mm/sec CNT100;
   1:  PR[GP1:91,1] = PR[GP1:90,1] + 56.741;
   1:  PR[GP1:91,2] = PR[GP1:90,2] + -13.564;
   1:L PR[91] R[100]mm/sec CNT100;
   1:  PR[GP1:91,1] = PR[GP1:90,1] + 58.961;
   1:  PR[GP1:91,2] = PR[GP1:90,2] + -1.308;
   1:L PR[91] R[100]mm/sec CNT100;
   1:  PR[GP1:91,1] = PR[GP1:90,1] + 59.159;
   1:  PR[GP1:91,2] = PR[GP1:90,2] + -0.078;
   1:L PR[91] R[100]mm/sec CNT100;
   1:  PR[GP1:91,1] = PR[GP1:90,1] + 57.222;
   1:  PR[GP1:91,2] = PR[GP1:90,2] + 10.581;
   1:L PR[91] R[100]mm/sec CNT100;
   1:  PR[GP1:91,1] = PR[GP1:90,1] + 57.036;
   1:  PR[GP1:91,2] = PR[GP1:90,2] + 11.828;
   1:L PR[91] R[100]mm/sec CNT100;
   1:  PR[GP1:91,1] = PR[GP1:90,1] + 56.743;
   1:  PR[GP1:91,2] = PR[GP1:90,2] + 13.415;
   1:L PR[91] R[100]mm/sec CNT100;
   1:  PR[GP1:91,1] = PR[GP1:90,1] + 50.806;
   1:  PR[GP1:91,2] = PR[GP1:90,2] + 23.440;
   1:L PR[91] R[100]mm/sec CNT100;
   1:  PR[GP1:91,1] = PR[GP1:90,1] + 49.612;
   1:  PR[GP1:91,2] = PR[GP1:90,2] + 25.414;
   1:L PR[91] R[100]mm/sec CNT100;
   1:  PR[GP1:91,1] = PR[GP1:90,1] + 41.112;
   1:  PR[GP1:91,2] = PR[GP1:90,2] + 32.437;
   1:L PR[91] R[100]mm/sec CNT100;
   1:  PR[GP1:91,1] = PR[GP1:90,1] + 38.519;
   1:  PR[GP1:91,2] = PR[GP1:90,2] + 34.490;
   1:L PR[91] R[100]mm/sec CNT100;
   1:  PR[GP1:91,1] = PR[GP1:90,1] + 28.935;
   1:  PR[GP1:91,2] = PR[GP1:90,2] + 38.024;
   1:L PR[91] R[100]mm/sec CNT100;
   1:  PR[GP1:91,1] = PR[GP1:90,1] + 24.689;
   1:  PR[GP1:91,2] = PR[GP1:90,2] + 39.417;
   1:L PR[91] R[100]mm/sec CNT100;
   1:  PR[GP1:91,1] = PR[GP1:90,1] + 15.416;
   1:  PR[GP1:91,2] = PR[GP1:90,2] + 39.585;
   1:L PR[91] R[100]mm/sec CNT100;
   1:  PR[GP1:91,1] = PR[GP1:90,1] + 9.780;
   1:  PR[GP1:91,2] = PR[GP1:90,2] + 39.383;
   1:L PR[91] R[100]mm/sec CNT100;
   1:  PR[GP1:91,1] = PR[GP1:90,1] + 1.921;
   1:  PR[GP1:91,2] = PR[GP1:90,2] + 36.956;
   1:L PR[91] R[100]mm/sec CNT100;
   1:  ! -- Layer/Ebene 135 -- !;
   1:  PR[91] = PR[90];
   1:  PR[GP1:91,1] = PR[GP1:90,1] + -1.684;
   1:  PR[GP1:91,2] = PR[GP1:90,2] + 37.130;
   1:  PR[GP1:91,3] = PR[GP1:90,3] + 82.655;
   1:L PR[91] R[100]mm/sec CNT100;
   1:  PR[GP1:91,1] = PR[GP1:90,1] + -9.271;
   1:  PR[GP1:91,2] = PR[GP1:90,2] + 39.472;
   1:L PR[91] R[100]mm/sec CNT100;
   1:  PR[GP1:91,1] = PR[GP1:90,1] + -15.242;
   1:  PR[GP1:91,2] = PR[GP1:90,2] + 39.686;
   1:L PR[91] R[100]mm/sec CNT100;
   1:  PR[GP1:91,1] = PR[GP1:90,1] + -24.216;
   1:  PR[GP1:91,2] = PR[GP1:90,2] + 39.522;
   1:L PR[91] R[100]mm/sec CNT100;
   1:  PR[GP1:91,1] = PR[GP1:90,1] + -28.792;
   1:  PR[GP1:91,2] = PR[GP1:90,2] + 38.022;
   1:L PR[91] R[100]mm/sec CNT100;
   1:  PR[GP1:91,1] = PR[GP1:90,1] + -38.085;
   1:  PR[GP1:91,2] = PR[GP1:90,2] + 34.592;
   1:L PR[91] R[100]mm/sec CNT100;
   1:  PR[GP1:91,1] = PR[GP1:90,1] + -40.960;
   1:  PR[GP1:91,2] = PR[GP1:90,2] + 32.317;
   1:L PR[91] R[100]mm/sec CNT100;
   1:  PR[GP1:91,1] = PR[GP1:90,1] + -49.215;
   1:  PR[GP1:91,2] = PR[GP1:90,2] + 25.503;
   1:L PR[91] R[100]mm/sec CNT100;
   1:  PR[GP1:91,1] = PR[GP1:90,1] + -50.601;
   1:  PR[GP1:91,2] = PR[GP1:90,2] + 23.212;
   1:L PR[91] R[100]mm/sec CNT100;
   1:  PR[GP1:91,1] = PR[GP1:90,1] + -56.371;
   1:  PR[GP1:91,2] = PR[GP1:90,2] + 13.447;
   1:L PR[91] R[100]mm/sec CNT100;
   1:  PR[GP1:91,1] = PR[GP1:90,1] + -58.528;
   1:  PR[GP1:91,2] = PR[GP1:90,2] + 1.552;
   1:L PR[91] R[100]mm/sec CNT100;
   1:  PR[GP1:91,1] = PR[GP1:90,1] + -58.788;
   1:  PR[GP1:91,2] = PR[GP1:90,2] + -0.066;
   1:L PR[91] R[100]mm/sec CNT100;
   1:  PR[GP1:91,1] = PR[GP1:90,1] + -56.959;
   1:  PR[GP1:91,2] = PR[GP1:90,2] + -10.115;
   1:L PR[91] R[100]mm/sec CNT100;
   1:  PR[GP1:91,1] = PR[GP1:90,1] + -56.732;
   1:  PR[GP1:91,2] = PR[GP1:90,2] + -11.633;
   1:L PR[91] R[100]mm/sec CNT100;
   1:  PR[GP1:91,1] = PR[GP1:90,1] + -56.370;
   1:  PR[GP1:91,2] = PR[GP1:90,2] + -13.593;
   1:L PR[91] R[100]mm/sec CNT100;
   1:  PR[GP1:91,1] = PR[GP1:90,1] + -50.596;
   1:  PR[GP1:91,2] = PR[GP1:90,2] + -23.361;
   1:L PR[91] R[100]mm/sec CNT100;
   1:  PR[GP1:91,1] = PR[GP1:90,1] + -49.211;
   1:  PR[GP1:91,2] = PR[GP1:90,2] + -25.653;
   1:L PR[91] R[100]mm/sec CNT100;
   1:  PR[GP1:91,1] = PR[GP1:90,1] + -40.952;
   1:  PR[GP1:91,2] = PR[GP1:90,2] + -32.465;
   1:L PR[91] R[100]mm/sec CNT100;
   1:  PR[GP1:91,1] = PR[GP1:90,1] + -38.077;
   1:  PR[GP1:91,2] = PR[GP1:90,2] + -34.740;
   1:L PR[91] R[100]mm/sec CNT100;
   1:  PR[GP1:91,1] = PR[GP1:90,1] + -28.781;
   1:  PR[GP1:91,2] = PR[GP1:90,2] + -38.167;
   1:L PR[91] R[100]mm/sec CNT100;
   1:  PR[GP1:91,1] = PR[GP1:90,1] + -24.205;
   1:  PR[GP1:91,2] = PR[GP1:90,2] + -39.668;
   1:L PR[91] R[100]mm/sec CNT100;
   1:  PR[GP1:91,1] = PR[GP1:90,1] + -15.231;
   1:  PR[GP1:91,2] = PR[GP1:90,2] + -39.828;
   1:L PR[91] R[100]mm/sec CNT100;
   1:  PR[GP1:91,1] = PR[GP1:90,1] + -9.262;
   1:  PR[GP1:91,2] = PR[GP1:90,2] + -39.615;
   1:L PR[91] R[100]mm/sec CNT100;
   1:  PR[GP1:91,1] = PR[GP1:90,1] + -1.686;
   1:  PR[GP1:91,2] = PR[GP1:90,2] + -37.259;
   1:L PR[91] R[100]mm/sec CNT100;
   1:  PR[GP1:91,1] = PR[GP1:90,1] + 1.897;
   1:  PR[GP1:91,2] = PR[GP1:90,2] + -37.258;
   1:L PR[91] R[100]mm/sec CNT100;
   1:  PR[GP1:91,1] = PR[GP1:90,1] + 9.474;
   1:  PR[GP1:91,2] = PR[GP1:90,2] + -39.614;
   1:L PR[91] R[100]mm/sec CNT100;
   1:  PR[GP1:91,1] = PR[GP1:90,1] + 15.443;
   1:  PR[GP1:91,2] = PR[GP1:90,2] + -39.827;
   1:L PR[91] R[100]mm/sec CNT100;
   1:  PR[GP1:91,1] = PR[GP1:90,1] + 24.417;
   1:  PR[GP1:91,2] = PR[GP1:90,2] + -39.669;
   1:L PR[91] R[100]mm/sec CNT100;
   1:  PR[GP1:91,1] = PR[GP1:90,1] + 28.993;
   1:  PR[GP1:91,2] = PR[GP1:90,2] + -38.167;
   1:L PR[91] R[100]mm/sec CNT100;
   1:  PR[GP1:91,1] = PR[GP1:90,1] + 38.289;
   1:  PR[GP1:91,2] = PR[GP1:90,2] + -34.743;
   1:L PR[91] R[100]mm/sec CNT100;
   1:  PR[GP1:91,1] = PR[GP1:90,1] + 41.164;
   1:  PR[GP1:91,2] = PR[GP1:90,2] + -32.467;
   1:L PR[91] R[100]mm/sec CNT100;
   1:  PR[GP1:91,1] = PR[GP1:90,1] + 49.423;
   1:  PR[GP1:91,2] = PR[GP1:90,2] + -25.647;
   1:L PR[91] R[100]mm/sec CNT100;
   1:  PR[GP1:91,1] = PR[GP1:90,1] + 50.809;
   1:  PR[GP1:91,2] = PR[GP1:90,2] + -23.356;
   1:L PR[91] R[100]mm/sec CNT100;
   1:  PR[GP1:91,1] = PR[GP1:90,1] + 56.583;
   1:  PR[GP1:91,2] = PR[GP1:90,2] + -13.610;
   1:L PR[91] R[100]mm/sec CNT100;
   1:  PR[GP1:91,1] = PR[GP1:90,1] + 58.741;
   1:  PR[GP1:91,2] = PR[GP1:90,2] + -1.696;
   1:L PR[91] R[100]mm/sec CNT100;
   1:  PR[GP1:91,1] = PR[GP1:90,1] + 59.002;
   1:  PR[GP1:91,2] = PR[GP1:90,2] + -0.078;
   1:L PR[91] R[100]mm/sec CNT100;
   1:  PR[GP1:91,1] = PR[GP1:90,1] + 57.173;
   1:  PR[GP1:91,2] = PR[GP1:90,2] + 9.982;
   1:L PR[91] R[100]mm/sec CNT100;
   1:  PR[GP1:91,1] = PR[GP1:90,1] + 56.946;
   1:  PR[GP1:91,2] = PR[GP1:90,2] + 11.502;
   1:L PR[91] R[100]mm/sec CNT100;
   1:  PR[GP1:91,1] = PR[GP1:90,1] + 56.585;
   1:  PR[GP1:91,2] = PR[GP1:90,2] + 13.462;
   1:L PR[91] R[100]mm/sec CNT100;
   1:  PR[GP1:91,1] = PR[GP1:90,1] + 50.813;
   1:  PR[GP1:91,2] = PR[GP1:90,2] + 23.207;
   1:L PR[91] R[100]mm/sec CNT100;
   1:  PR[GP1:91,1] = PR[GP1:90,1] + 49.428;
   1:  PR[GP1:91,2] = PR[GP1:90,2] + 25.498;
   1:L PR[91] R[100]mm/sec CNT100;
   1:  PR[GP1:91,1] = PR[GP1:90,1] + 41.172;
   1:  PR[GP1:91,2] = PR[GP1:90,2] + 32.319;
   1:L PR[91] R[100]mm/sec CNT100;
   1:  PR[GP1:91,1] = PR[GP1:90,1] + 38.297;
   1:  PR[GP1:91,2] = PR[GP1:90,2] + 34.594;
   1:L PR[91] R[100]mm/sec CNT100;
   1:  PR[GP1:91,1] = PR[GP1:90,1] + 29.003;
   1:  PR[GP1:91,2] = PR[GP1:90,2] + 38.022;
   1:L PR[91] R[100]mm/sec CNT100;
   1:  PR[GP1:91,1] = PR[GP1:90,1] + 24.428;
   1:  PR[GP1:91,2] = PR[GP1:90,2] + 39.523;
   1:L PR[91] R[100]mm/sec CNT100;
   1:  PR[GP1:91,1] = PR[GP1:90,1] + 15.454;
   1:  PR[GP1:91,2] = PR[GP1:90,2] + 39.685;
   1:L PR[91] R[100]mm/sec CNT100;
   1:  PR[GP1:91,1] = PR[GP1:90,1] + 9.483;
   1:  PR[GP1:91,2] = PR[GP1:90,2] + 39.471;
   1:L PR[91] R[100]mm/sec CNT100;
   1:  PR[GP1:91,1] = PR[GP1:90,1] + 1.896;
   1:  PR[GP1:91,2] = PR[GP1:90,2] + 37.129;
   1:L PR[91] R[100]mm/sec CNT100;
   1:  ! -- Layer/Ebene 136 -- !;
   1:  PR[91] = PR[90];
   1:  PR[GP1:91,1] = PR[GP1:90,1] + -1.658;
   1:  PR[GP1:91,2] = PR[GP1:90,2] + 37.303;
   1:  PR[GP1:91,3] = PR[GP1:90,3] + 83.265;
   1:L PR[91] R[100]mm/sec CNT100;
   1:  PR[GP1:91,1] = PR[GP1:90,1] + -8.973;
   1:  PR[GP1:91,2] = PR[GP1:90,2] + 39.560;
   1:L PR[91] R[100]mm/sec CNT100;
   1:  PR[GP1:91,1] = PR[GP1:90,1] + -15.280;
   1:  PR[GP1:91,2] = PR[GP1:90,2] + 39.787;
   1:L PR[91] R[100]mm/sec CNT100;
   1:  PR[GP1:91,1] = PR[GP1:90,1] + -23.955;
   1:  PR[GP1:91,2] = PR[GP1:90,2] + 39.628;
   1:L PR[91] R[100]mm/sec CNT100;
   1:  PR[GP1:91,1] = PR[GP1:90,1] + -28.860;
   1:  PR[GP1:91,2] = PR[GP1:90,2] + 38.020;
   1:L PR[91] R[100]mm/sec CNT100;
   1:  PR[GP1:91,1] = PR[GP1:90,1] + -37.864;
   1:  PR[GP1:91,2] = PR[GP1:90,2] + 34.697;
   1:L PR[91] R[100]mm/sec CNT100;
   1:  PR[GP1:91,1] = PR[GP1:90,1] + -41.020;
   1:  PR[GP1:91,2] = PR[GP1:90,2] + 32.199;
   1:L PR[91] R[100]mm/sec CNT100;
   1:  PR[GP1:91,1] = PR[GP1:90,1] + -49.030;
   1:  PR[GP1:91,2] = PR[GP1:90,2] + 25.588;
   1:L PR[91] R[100]mm/sec CNT100;
   1:  PR[GP1:91,1] = PR[GP1:90,1] + -50.608;
   1:  PR[GP1:91,2] = PR[GP1:90,2] + 22.979;
   1:L PR[91] R[100]mm/sec CNT100;
   1:  PR[GP1:91,1] = PR[GP1:90,1] + -56.213;
   1:  PR[GP1:91,2] = PR[GP1:90,2] + 13.494;
   1:L PR[91] R[100]mm/sec CNT100;
   1:  PR[GP1:91,1] = PR[GP1:90,1] + -58.307;
   1:  PR[GP1:91,2] = PR[GP1:90,2] + 1.940;
   1:L PR[91] R[100]mm/sec CNT100;
   1:  PR[GP1:91,1] = PR[GP1:90,1] + -58.631;
   1:  PR[GP1:91,2] = PR[GP1:90,2] + -0.066;
   1:L PR[91] R[100]mm/sec CNT100;
   1:  PR[GP1:91,1] = PR[GP1:90,1] + -56.910;
   1:  PR[GP1:91,2] = PR[GP1:90,2] + -9.517;
   1:L PR[91] R[100]mm/sec CNT100;
   1:  PR[GP1:91,1] = PR[GP1:90,1] + -56.642;
   1:  PR[GP1:91,2] = PR[GP1:90,2] + -11.308;
   1:L PR[91] R[100]mm/sec CNT100;
   1:  PR[GP1:91,1] = PR[GP1:90,1] + -56.212;
   1:  PR[GP1:91,2] = PR[GP1:90,2] + -13.640;
   1:L PR[91] R[100]mm/sec CNT100;
   1:  PR[GP1:91,1] = PR[GP1:90,1] + -50.603;
   1:  PR[GP1:91,2] = PR[GP1:90,2] + -23.128;
   1:L PR[91] R[100]mm/sec CNT100;
   1:  PR[GP1:91,1] = PR[GP1:90,1] + -49.026;
   1:  PR[GP1:91,2] = PR[GP1:90,2] + -25.737;
   1:L PR[91] R[100]mm/sec CNT100;
   1:  PR[GP1:91,1] = PR[GP1:90,1] + -41.012;
   1:  PR[GP1:91,2] = PR[GP1:90,2] + -32.347;
   1:L PR[91] R[100]mm/sec CNT100;
   1:  PR[GP1:91,1] = PR[GP1:90,1] + -37.856;
   1:  PR[GP1:91,2] = PR[GP1:90,2] + -34.845;
   1:L PR[91] R[100]mm/sec CNT100;
   1:  PR[GP1:91,1] = PR[GP1:90,1] + -28.850;
   1:  PR[GP1:91,2] = PR[GP1:90,2] + -38.165;
   1:L PR[91] R[100]mm/sec CNT100;
   1:  PR[GP1:91,1] = PR[GP1:90,1] + -23.944;
   1:  PR[GP1:91,2] = PR[GP1:90,2] + -39.774;
   1:L PR[91] R[100]mm/sec CNT100;
   1:  PR[GP1:91,1] = PR[GP1:90,1] + -15.269;
   1:  PR[GP1:91,2] = PR[GP1:90,2] + -39.928;
   1:L PR[91] R[100]mm/sec CNT100;
   1:  PR[GP1:91,1] = PR[GP1:90,1] + -8.965;
   1:  PR[GP1:91,2] = PR[GP1:90,2] + -39.703;
   1:L PR[91] R[100]mm/sec CNT100;
   1:  PR[GP1:91,1] = PR[GP1:90,1] + -1.661;
   1:  PR[GP1:91,2] = PR[GP1:90,2] + -37.433;
   1:L PR[91] R[100]mm/sec CNT100;
   1:  PR[GP1:91,1] = PR[GP1:90,1] + 1.872;
   1:  PR[GP1:91,2] = PR[GP1:90,2] + -37.432;
   1:L PR[91] R[100]mm/sec CNT100;
   1:  PR[GP1:91,1] = PR[GP1:90,1] + 9.177;
   1:  PR[GP1:91,2] = PR[GP1:90,2] + -39.703;
   1:L PR[91] R[100]mm/sec CNT100;
   1:  PR[GP1:91,1] = PR[GP1:90,1] + 15.482;
   1:  PR[GP1:91,2] = PR[GP1:90,2] + -39.928;
   1:L PR[91] R[100]mm/sec CNT100;
   1:  PR[GP1:91,1] = PR[GP1:90,1] + 24.157;
   1:  PR[GP1:91,2] = PR[GP1:90,2] + -39.775;
   1:L PR[91] R[100]mm/sec CNT100;
   1:  PR[GP1:91,1] = PR[GP1:90,1] + 29.062;
   1:  PR[GP1:91,2] = PR[GP1:90,2] + -38.165;
   1:L PR[91] R[100]mm/sec CNT100;
   1:  PR[GP1:91,1] = PR[GP1:90,1] + 38.068;
   1:  PR[GP1:91,2] = PR[GP1:90,2] + -34.848;
   1:L PR[91] R[100]mm/sec CNT100;
   1:  PR[GP1:91,1] = PR[GP1:90,1] + 41.224;
   1:  PR[GP1:91,2] = PR[GP1:90,2] + -32.349;
   1:L PR[91] R[100]mm/sec CNT100;
   1:  PR[GP1:91,1] = PR[GP1:90,1] + 49.239;
   1:  PR[GP1:91,2] = PR[GP1:90,2] + -25.731;
   1:L PR[91] R[100]mm/sec CNT100;
   1:  PR[GP1:91,1] = PR[GP1:90,1] + 50.816;
   1:  PR[GP1:91,2] = PR[GP1:90,2] + -23.123;
   1:L PR[91] R[100]mm/sec CNT100;
   1:  PR[GP1:91,1] = PR[GP1:90,1] + 56.424;
   1:  PR[GP1:91,2] = PR[GP1:90,2] + -13.657;
   1:L PR[91] R[100]mm/sec CNT100;
   1:  PR[GP1:91,1] = PR[GP1:90,1] + 58.521;
   1:  PR[GP1:91,2] = PR[GP1:90,2] + -2.085;
   1:L PR[91] R[100]mm/sec CNT100;
   1:  PR[GP1:91,1] = PR[GP1:90,1] + 58.844;
   1:  PR[GP1:91,2] = PR[GP1:90,2] + -0.078;
   1:L PR[91] R[100]mm/sec CNT100;
   1:  PR[GP1:91,1] = PR[GP1:90,1] + 57.125;
   1:  PR[GP1:91,2] = PR[GP1:90,2] + 9.383;
   1:L PR[91] R[100]mm/sec CNT100;
   1:  PR[GP1:91,1] = PR[GP1:90,1] + 56.856;
   1:  PR[GP1:91,2] = PR[GP1:90,2] + 11.176;
   1:L PR[91] R[100]mm/sec CNT100;
   1:  PR[GP1:91,1] = PR[GP1:90,1] + 56.426;
   1:  PR[GP1:91,2] = PR[GP1:90,2] + 13.509;
   1:L PR[91] R[100]mm/sec CNT100;
   1:  PR[GP1:91,1] = PR[GP1:90,1] + 50.820;
   1:  PR[GP1:91,2] = PR[GP1:90,2] + 22.975;
   1:L PR[91] R[100]mm/sec CNT100;
   1:  PR[GP1:91,1] = PR[GP1:90,1] + 49.243;
   1:  PR[GP1:91,2] = PR[GP1:90,2] + 25.582;
   1:L PR[91] R[100]mm/sec CNT100;
   1:  PR[GP1:91,1] = PR[GP1:90,1] + 41.232;
   1:  PR[GP1:91,2] = PR[GP1:90,2] + 32.201;
   1:L PR[91] R[100]mm/sec CNT100;
   1:  PR[GP1:91,1] = PR[GP1:90,1] + 38.076;
   1:  PR[GP1:91,2] = PR[GP1:90,2] + 34.699;
   1:L PR[91] R[100]mm/sec CNT100;
   1:  PR[GP1:91,1] = PR[GP1:90,1] + 29.072;
   1:  PR[GP1:91,2] = PR[GP1:90,2] + 38.020;
   1:L PR[91] R[100]mm/sec CNT100;
   1:  PR[GP1:91,1] = PR[GP1:90,1] + 24.167;
   1:  PR[GP1:91,2] = PR[GP1:90,2] + 39.629;
   1:L PR[91] R[100]mm/sec CNT100;
   1:  PR[GP1:91,1] = PR[GP1:90,1] + 15.493;
   1:  PR[GP1:91,2] = PR[GP1:90,2] + 39.786;
   1:L PR[91] R[100]mm/sec CNT100;
   1:  PR[GP1:91,1] = PR[GP1:90,1] + 9.186;
   1:  PR[GP1:91,2] = PR[GP1:90,2] + 39.560;
   1:L PR[91] R[100]mm/sec CNT100;
   1:  PR[GP1:91,1] = PR[GP1:90,1] + 1.871;
   1:  PR[GP1:91,2] = PR[GP1:90,2] + 37.302;
   1:L PR[91] R[100]mm/sec CNT100;
   1:  ! -- Layer/Ebene 137 -- !;
   1:  PR[91] = PR[90];
   1:  PR[GP1:91,1] = PR[GP1:90,1] + -1.633;
   1:  PR[GP1:91,2] = PR[GP1:90,2] + 37.477;
   1:  PR[GP1:91,3] = PR[GP1:90,3] + 83.875;
   1:L PR[91] R[100]mm/sec CNT100;
   1:  PR[GP1:91,1] = PR[GP1:90,1] + -8.676;
   1:  PR[GP1:91,2] = PR[GP1:90,2] + 39.649;
   1:L PR[91] R[100]mm/sec CNT100;
   1:  PR[GP1:91,1] = PR[GP1:90,1] + -15.319;
   1:  PR[GP1:91,2] = PR[GP1:90,2] + 39.887;
   1:L PR[91] R[100]mm/sec CNT100;
   1:  PR[GP1:91,1] = PR[GP1:90,1] + -23.693;
   1:  PR[GP1:91,2] = PR[GP1:90,2] + 39.734;
   1:L PR[91] R[100]mm/sec CNT100;
   1:  PR[GP1:91,1] = PR[GP1:90,1] + -28.928;
   1:  PR[GP1:91,2] = PR[GP1:90,2] + 38.018;
   1:L PR[91] R[100]mm/sec CNT100;
   1:  PR[GP1:91,1] = PR[GP1:90,1] + -37.642;
   1:  PR[GP1:91,2] = PR[GP1:90,2] + 34.802;
   1:L PR[91] R[100]mm/sec CNT100;
   1:  PR[GP1:91,1] = PR[GP1:90,1] + -41.080;
   1:  PR[GP1:91,2] = PR[GP1:90,2] + 32.082;
   1:L PR[91] R[100]mm/sec CNT100;
   1:  PR[GP1:91,1] = PR[GP1:90,1] + -48.846;
   1:  PR[GP1:91,2] = PR[GP1:90,2] + 25.672;
   1:L PR[91] R[100]mm/sec CNT100;
   1:  PR[GP1:91,1] = PR[GP1:90,1] + -50.615;
   1:  PR[GP1:91,2] = PR[GP1:90,2] + 22.746;
   1:L PR[91] R[100]mm/sec CNT100;
   1:  PR[GP1:91,1] = PR[GP1:90,1] + -56.054;
   1:  PR[GP1:91,2] = PR[GP1:90,2] + 13.541;
   1:L PR[91] R[100]mm/sec CNT100;
   1:  PR[GP1:91,1] = PR[GP1:90,1] + -58.087;
   1:  PR[GP1:91,2] = PR[GP1:90,2] + 2.328;
   1:L PR[91] R[100]mm/sec CNT100;
   1:  PR[GP1:91,1] = PR[GP1:90,1] + -58.473;
   1:  PR[GP1:91,2] = PR[GP1:90,2] + -0.066;
   1:L PR[91] R[100]mm/sec CNT100;
   1:  PR[GP1:91,1] = PR[GP1:90,1] + -56.862;
   1:  PR[GP1:91,2] = PR[GP1:90,2] + -8.918;
   1:L PR[91] R[100]mm/sec CNT100;
   1:  PR[GP1:91,1] = PR[GP1:90,1] + -56.553;
   1:  PR[GP1:91,2] = PR[GP1:90,2] + -10.982;
   1:L PR[91] R[100]mm/sec CNT100;
   1:  PR[GP1:91,1] = PR[GP1:90,1] + -56.053;
   1:  PR[GP1:91,2] = PR[GP1:90,2] + -13.688;
   1:L PR[91] R[100]mm/sec CNT100;
   1:  PR[GP1:91,1] = PR[GP1:90,1] + -50.610;
   1:  PR[GP1:91,2] = PR[GP1:90,2] + -22.895;
   1:L PR[91] R[100]mm/sec CNT100;
   1:  PR[GP1:91,1] = PR[GP1:90,1] + -48.842;
   1:  PR[GP1:91,2] = PR[GP1:90,2] + -25.820;
   1:L PR[91] R[100]mm/sec CNT100;
   1:  PR[GP1:91,1] = PR[GP1:90,1] + -41.072;
   1:  PR[GP1:91,2] = PR[GP1:90,2] + -32.230;
   1:L PR[91] R[100]mm/sec CNT100;
   1:  PR[GP1:91,1] = PR[GP1:90,1] + -37.635;
   1:  PR[GP1:91,2] = PR[GP1:90,2] + -34.950;
   1:L PR[91] R[100]mm/sec CNT100;
   1:  PR[GP1:91,1] = PR[GP1:90,1] + -28.919;
   1:  PR[GP1:91,2] = PR[GP1:90,2] + -38.163;
   1:L PR[91] R[100]mm/sec CNT100;
   1:  PR[GP1:91,1] = PR[GP1:90,1] + -23.683;
   1:  PR[GP1:91,2] = PR[GP1:90,2] + -39.880;
   1:L PR[91] R[100]mm/sec CNT100;
   1:  PR[GP1:91,1] = PR[GP1:90,1] + -15.308;
   1:  PR[GP1:91,2] = PR[GP1:90,2] + -40.029;
   1:L PR[91] R[100]mm/sec CNT100;
   1:  PR[GP1:91,1] = PR[GP1:90,1] + -8.668;
   1:  PR[GP1:91,2] = PR[GP1:90,2] + -39.792;
   1:L PR[91] R[100]mm/sec CNT100;
   1:  PR[GP1:91,1] = PR[GP1:90,1] + -1.635;
   1:  PR[GP1:91,2] = PR[GP1:90,2] + -37.606;
   1:L PR[91] R[100]mm/sec CNT100;
   1:  PR[GP1:91,1] = PR[GP1:90,1] + 1.847;
   1:  PR[GP1:91,2] = PR[GP1:90,2] + -37.605;
   1:L PR[91] R[100]mm/sec CNT100;
   1:  PR[GP1:91,1] = PR[GP1:90,1] + 8.880;
   1:  PR[GP1:91,2] = PR[GP1:90,2] + -39.792;
   1:L PR[91] R[100]mm/sec CNT100;
   1:  PR[GP1:91,1] = PR[GP1:90,1] + 15.521;
   1:  PR[GP1:91,2] = PR[GP1:90,2] + -40.028;
   1:L PR[91] R[100]mm/sec CNT100;
   1:  PR[GP1:91,1] = PR[GP1:90,1] + 23.896;
   1:  PR[GP1:91,2] = PR[GP1:90,2] + -39.881;
   1:L PR[91] R[100]mm/sec CNT100;
   1:  PR[GP1:91,1] = PR[GP1:90,1] + 29.131;
   1:  PR[GP1:91,2] = PR[GP1:90,2] + -38.163;
   1:L PR[91] R[100]mm/sec CNT100;
   1:  PR[GP1:91,1] = PR[GP1:90,1] + 37.847;
   1:  PR[GP1:91,2] = PR[GP1:90,2] + -34.952;
   1:L PR[91] R[100]mm/sec CNT100;
   1:  PR[GP1:91,1] = PR[GP1:90,1] + 41.285;
   1:  PR[GP1:91,2] = PR[GP1:90,2] + -32.231;
   1:L PR[91] R[100]mm/sec CNT100;
   1:  PR[GP1:91,1] = PR[GP1:90,1] + 49.054;
   1:  PR[GP1:91,2] = PR[GP1:90,2] + -25.815;
   1:L PR[91] R[100]mm/sec CNT100;
   1:  PR[GP1:91,1] = PR[GP1:90,1] + 50.823;
   1:  PR[GP1:91,2] = PR[GP1:90,2] + -22.891;
   1:L PR[91] R[100]mm/sec CNT100;
   1:  PR[GP1:91,1] = PR[GP1:90,1] + 56.266;
   1:  PR[GP1:91,2] = PR[GP1:90,2] + -13.704;
   1:L PR[91] R[100]mm/sec CNT100;
   1:  PR[GP1:91,1] = PR[GP1:90,1] + 58.300;
   1:  PR[GP1:91,2] = PR[GP1:90,2] + -2.473;
   1:L PR[91] R[100]mm/sec CNT100;
   1:  PR[GP1:91,1] = PR[GP1:90,1] + 58.686;
   1:  PR[GP1:91,2] = PR[GP1:90,2] + -0.078;
   1:L PR[91] R[100]mm/sec CNT100;
   1:  PR[GP1:91,1] = PR[GP1:90,1] + 57.076;
   1:  PR[GP1:91,2] = PR[GP1:90,2] + 8.784;
   1:L PR[91] R[100]mm/sec CNT100;
   1:  PR[GP1:91,1] = PR[GP1:90,1] + 56.767;
   1:  PR[GP1:91,2] = PR[GP1:90,2] + 10.850;
   1:L PR[91] R[100]mm/sec CNT100;
   1:  PR[GP1:91,1] = PR[GP1:90,1] + 56.268;
   1:  PR[GP1:91,2] = PR[GP1:90,2] + 13.556;
   1:L PR[91] R[100]mm/sec CNT100;
   1:  PR[GP1:91,1] = PR[GP1:90,1] + 50.827;
   1:  PR[GP1:91,2] = PR[GP1:90,2] + 22.742;
   1:L PR[91] R[100]mm/sec CNT100;
   1:  PR[GP1:91,1] = PR[GP1:90,1] + 49.058;
   1:  PR[GP1:91,2] = PR[GP1:90,2] + 25.666;
   1:L PR[91] R[100]mm/sec CNT100;
   1:  PR[GP1:91,1] = PR[GP1:90,1] + 41.292;
   1:  PR[GP1:91,2] = PR[GP1:90,2] + 32.084;
   1:L PR[91] R[100]mm/sec CNT100;
   1:  PR[GP1:91,1] = PR[GP1:90,1] + 37.854;
   1:  PR[GP1:91,2] = PR[GP1:90,2] + 34.804;
   1:L PR[91] R[100]mm/sec CNT100;
   1:  PR[GP1:91,1] = PR[GP1:90,1] + 29.140;
   1:  PR[GP1:91,2] = PR[GP1:90,2] + 38.018;
   1:L PR[91] R[100]mm/sec CNT100;
   1:  PR[GP1:91,1] = PR[GP1:90,1] + 23.905;
   1:  PR[GP1:91,2] = PR[GP1:90,2] + 39.735;
   1:L PR[91] R[100]mm/sec CNT100;
   1:  PR[GP1:91,1] = PR[GP1:90,1] + 15.531;
   1:  PR[GP1:91,2] = PR[GP1:90,2] + 39.887;
   1:L PR[91] R[100]mm/sec CNT100;
   1:  PR[GP1:91,1] = PR[GP1:90,1] + 8.888;
   1:  PR[GP1:91,2] = PR[GP1:90,2] + 39.649;
   1:L PR[91] R[100]mm/sec CNT100;
   1:  PR[GP1:91,1] = PR[GP1:90,1] + 1.845;
   1:  PR[GP1:91,2] = PR[GP1:90,2] + 37.476;
   1:L PR[91] R[100]mm/sec CNT100;
   1:  ! -- Layer/Ebene 138 -- !;
   1:  PR[91] = PR[90];
   1:  PR[GP1:91,1] = PR[GP1:90,1] + -1.608;
   1:  PR[GP1:91,2] = PR[GP1:90,2] + 37.650;
   1:  PR[GP1:91,3] = PR[GP1:90,3] + 84.485;
   1:L PR[91] R[100]mm/sec CNT100;
   1:  PR[GP1:91,1] = PR[GP1:90,1] + -8.378;
   1:  PR[GP1:91,2] = PR[GP1:90,2] + 39.738;
   1:L PR[91] R[100]mm/sec CNT100;
   1:  PR[GP1:91,1] = PR[GP1:90,1] + -15.357;
   1:  PR[GP1:91,2] = PR[GP1:90,2] + 39.988;
   1:L PR[91] R[100]mm/sec CNT100;
   1:  PR[GP1:91,1] = PR[GP1:90,1] + -23.432;
   1:  PR[GP1:91,2] = PR[GP1:90,2] + 39.841;
   1:L PR[91] R[100]mm/sec CNT100;
   1:  PR[GP1:91,1] = PR[GP1:90,1] + -28.997;
   1:  PR[GP1:91,2] = PR[GP1:90,2] + 38.016;
   1:L PR[91] R[100]mm/sec CNT100;
   1:  PR[GP1:91,1] = PR[GP1:90,1] + -37.421;
   1:  PR[GP1:91,2] = PR[GP1:90,2] + 34.907;
   1:L PR[91] R[100]mm/sec CNT100;
   1:  PR[GP1:91,1] = PR[GP1:90,1] + -41.140;
   1:  PR[GP1:91,2] = PR[GP1:90,2] + 31.964;
   1:L PR[91] R[100]mm/sec CNT100;
   1:  PR[GP1:91,1] = PR[GP1:90,1] + -48.661;
   1:  PR[GP1:91,2] = PR[GP1:90,2] + 25.756;
   1:L PR[91] R[100]mm/sec CNT100;
   1:  PR[GP1:91,1] = PR[GP1:90,1] + -50.622;
   1:  PR[GP1:91,2] = PR[GP1:90,2] + 22.513;
   1:L PR[91] R[100]mm/sec CNT100;
   1:  PR[GP1:91,1] = PR[GP1:90,1] + -55.896;
   1:  PR[GP1:91,2] = PR[GP1:90,2] + 13.589;
   1:L PR[91] R[100]mm/sec CNT100;
   1:  PR[GP1:91,1] = PR[GP1:90,1] + -57.867;
   1:  PR[GP1:91,2] = PR[GP1:90,2] + 2.716;
   1:L PR[91] R[100]mm/sec CNT100;
   1:  PR[GP1:91,1] = PR[GP1:90,1] + -58.315;
   1:  PR[GP1:91,2] = PR[GP1:90,2] + -0.066;
   1:L PR[91] R[100]mm/sec CNT100;
   1:  PR[GP1:91,1] = PR[GP1:90,1] + -56.813;
   1:  PR[GP1:91,2] = PR[GP1:90,2] + -8.320;
   1:L PR[91] R[100]mm/sec CNT100;
   1:  PR[GP1:91,1] = PR[GP1:90,1] + -56.463;
   1:  PR[GP1:91,2] = PR[GP1:90,2] + -10.656;
   1:L PR[91] R[100]mm/sec CNT100;
   1:  PR[GP1:91,1] = PR[GP1:90,1] + -55.895;
   1:  PR[GP1:91,2] = PR[GP1:90,2] + -13.735;
   1:L PR[91] R[100]mm/sec CNT100;
   1:  PR[GP1:91,1] = PR[GP1:90,1] + -50.617;
   1:  PR[GP1:91,2] = PR[GP1:90,2] + -22.662;
   1:L PR[91] R[100]mm/sec CNT100;
   1:  PR[GP1:91,1] = PR[GP1:90,1] + -48.657;
   1:  PR[GP1:91,2] = PR[GP1:90,2] + -25.904;
   1:L PR[91] R[100]mm/sec CNT100;
   1:  PR[GP1:91,1] = PR[GP1:90,1] + -41.132;
   1:  PR[GP1:91,2] = PR[GP1:90,2] + -32.112;
   1:L PR[91] R[100]mm/sec CNT100;
   1:  PR[GP1:91,1] = PR[GP1:90,1] + -37.413;
   1:  PR[GP1:91,2] = PR[GP1:90,2] + -35.055;
   1:L PR[91] R[100]mm/sec CNT100;
   1:  PR[GP1:91,1] = PR[GP1:90,1] + -28.988;
   1:  PR[GP1:91,2] = PR[GP1:90,2] + -38.161;
   1:L PR[91] R[100]mm/sec CNT100;
   1:  PR[GP1:91,1] = PR[GP1:90,1] + -23.422;
   1:  PR[GP1:91,2] = PR[GP1:90,2] + -39.986;
   1:L PR[91] R[100]mm/sec CNT100;
   1:  PR[GP1:91,1] = PR[GP1:90,1] + -15.347;
   1:  PR[GP1:91,2] = PR[GP1:90,2] + -40.130;
   1:L PR[91] R[100]mm/sec CNT100;
   1:  PR[GP1:91,1] = PR[GP1:90,1] + -8.371;
   1:  PR[GP1:91,2] = PR[GP1:90,2] + -39.881;
   1:L PR[91] R[100]mm/sec CNT100;
   1:  PR[GP1:91,1] = PR[GP1:90,1] + -1.610;
   1:  PR[GP1:91,2] = PR[GP1:90,2] + -37.780;
   1:L PR[91] R[100]mm/sec CNT100;
   1:  PR[GP1:91,1] = PR[GP1:90,1] + 1.822;
   1:  PR[GP1:91,2] = PR[GP1:90,2] + -37.779;
   1:L PR[91] R[100]mm/sec CNT100;
   1:  PR[GP1:91,1] = PR[GP1:90,1] + 8.584;
   1:  PR[GP1:91,2] = PR[GP1:90,2] + -39.881;
   1:L PR[91] R[100]mm/sec CNT100;
   1:  PR[GP1:91,1] = PR[GP1:90,1] + 15.559;
   1:  PR[GP1:91,2] = PR[GP1:90,2] + -40.129;
   1:L PR[91] R[100]mm/sec CNT100;
   1:  PR[GP1:91,1] = PR[GP1:90,1] + 23.635;
   1:  PR[GP1:91,2] = PR[GP1:90,2] + -39.987;
   1:L PR[91] R[100]mm/sec CNT100;
   1:  PR[GP1:91,1] = PR[GP1:90,1] + 29.200;
   1:  PR[GP1:91,2] = PR[GP1:90,2] + -38.161;
   1:L PR[91] R[100]mm/sec CNT100;
   1:  PR[GP1:91,1] = PR[GP1:90,1] + 37.626;
   1:  PR[GP1:91,2] = PR[GP1:90,2] + -35.057;
   1:L PR[91] R[100]mm/sec CNT100;
   1:  PR[GP1:91,1] = PR[GP1:90,1] + 41.345;
   1:  PR[GP1:91,2] = PR[GP1:90,2] + -32.113;
   1:L PR[91] R[100]mm/sec CNT100;
   1:  PR[GP1:91,1] = PR[GP1:90,1] + 48.870;
   1:  PR[GP1:91,2] = PR[GP1:90,2] + -25.899;
   1:L PR[91] R[100]mm/sec CNT100;
   1:  PR[GP1:91,1] = PR[GP1:90,1] + 50.830;
   1:  PR[GP1:91,2] = PR[GP1:90,2] + -22.658;
   1:L PR[91] R[100]mm/sec CNT100;
   1:  PR[GP1:91,1] = PR[GP1:90,1] + 56.108;
   1:  PR[GP1:91,2] = PR[GP1:90,2] + -13.751;
   1:L PR[91] R[100]mm/sec CNT100;
   1:  PR[GP1:91,1] = PR[GP1:90,1] + 58.080;
   1:  PR[GP1:91,2] = PR[GP1:90,2] + -2.861;
   1:L PR[91] R[100]mm/sec CNT100;
   1:  PR[GP1:91,1] = PR[GP1:90,1] + 58.528;
   1:  PR[GP1:91,2] = PR[GP1:90,2] + -0.078;
   1:L PR[91] R[100]mm/sec CNT100;
   1:  PR[GP1:91,1] = PR[GP1:90,1] + 57.027;
   1:  PR[GP1:91,2] = PR[GP1:90,2] + 8.185;
   1:L PR[91] R[100]mm/sec CNT100;
   1:  PR[GP1:91,1] = PR[GP1:90,1] + 56.677;
   1:  PR[GP1:91,2] = PR[GP1:90,2] + 10.524;
   1:L PR[91] R[100]mm/sec CNT100;
   1:  PR[GP1:91,1] = PR[GP1:90,1] + 56.109;
   1:  PR[GP1:91,2] = PR[GP1:90,2] + 13.603;
   1:L PR[91] R[100]mm/sec CNT100;
   1:  PR[GP1:91,1] = PR[GP1:90,1] + 50.834;
   1:  PR[GP1:91,2] = PR[GP1:90,2] + 22.510;
   1:L PR[91] R[100]mm/sec CNT100;
   1:  PR[GP1:91,1] = PR[GP1:90,1] + 48.874;
   1:  PR[GP1:91,2] = PR[GP1:90,2] + 25.751;
   1:L PR[91] R[100]mm/sec CNT100;
   1:  PR[GP1:91,1] = PR[GP1:90,1] + 41.351;
   1:  PR[GP1:91,2] = PR[GP1:90,2] + 31.966;
   1:L PR[91] R[100]mm/sec CNT100;
   1:  PR[GP1:91,1] = PR[GP1:90,1] + 37.633;
   1:  PR[GP1:91,2] = PR[GP1:90,2] + 34.909;
   1:L PR[91] R[100]mm/sec CNT100;
   1:  PR[GP1:91,1] = PR[GP1:90,1] + 29.209;
   1:  PR[GP1:91,2] = PR[GP1:90,2] + 38.016;
   1:L PR[91] R[100]mm/sec CNT100;
   1:  PR[GP1:91,1] = PR[GP1:90,1] + 23.644;
   1:  PR[GP1:91,2] = PR[GP1:90,2] + 39.841;
   1:L PR[91] R[100]mm/sec CNT100;
   1:  PR[GP1:91,1] = PR[GP1:90,1] + 15.569;
   1:  PR[GP1:91,2] = PR[GP1:90,2] + 39.987;
   1:L PR[91] R[100]mm/sec CNT100;
   1:  PR[GP1:91,1] = PR[GP1:90,1] + 8.591;
   1:  PR[GP1:91,2] = PR[GP1:90,2] + 39.737;
   1:L PR[91] R[100]mm/sec CNT100;
   1:  PR[GP1:91,1] = PR[GP1:90,1] + 1.820;
   1:  PR[GP1:91,2] = PR[GP1:90,2] + 37.649;
   1:L PR[91] R[100]mm/sec CNT100;
   1:  ! -- Layer/Ebene 139 -- !;
   1:  PR[91] = PR[90];
   1:  PR[GP1:91,1] = PR[GP1:90,1] + -1.583;
   1:  PR[GP1:91,2] = PR[GP1:90,2] + 37.823;
   1:  PR[GP1:91,3] = PR[GP1:90,3] + 85.095;
   1:L PR[91] R[100]mm/sec CNT100;
   1:  PR[GP1:91,1] = PR[GP1:90,1] + -8.081;
   1:  PR[GP1:91,2] = PR[GP1:90,2] + 39.826;
   1:L PR[91] R[100]mm/sec CNT100;
   1:  PR[GP1:91,1] = PR[GP1:90,1] + -15.395;
   1:  PR[GP1:91,2] = PR[GP1:90,2] + 40.089;
   1:L PR[91] R[100]mm/sec CNT100;
   1:  PR[GP1:91,1] = PR[GP1:90,1] + -23.171;
   1:  PR[GP1:91,2] = PR[GP1:90,2] + 39.947;
   1:L PR[91] R[100]mm/sec CNT100;
   1:  PR[GP1:91,1] = PR[GP1:90,1] + -29.065;
   1:  PR[GP1:91,2] = PR[GP1:90,2] + 38.014;
   1:L PR[91] R[100]mm/sec CNT100;
   1:  PR[GP1:91,1] = PR[GP1:90,1] + -37.199;
   1:  PR[GP1:91,2] = PR[GP1:90,2] + 35.012;
   1:L PR[91] R[100]mm/sec CNT100;
   1:  PR[GP1:91,1] = PR[GP1:90,1] + -41.199;
   1:  PR[GP1:91,2] = PR[GP1:90,2] + 31.846;
   1:L PR[91] R[100]mm/sec CNT100;
   1:  PR[GP1:91,1] = PR[GP1:90,1] + -48.476;
   1:  PR[GP1:91,2] = PR[GP1:90,2] + 25.840;
   1:L PR[91] R[100]mm/sec CNT100;
   1:  PR[GP1:91,1] = PR[GP1:90,1] + -50.628;
   1:  PR[GP1:91,2] = PR[GP1:90,2] + 22.281;
   1:L PR[91] R[100]mm/sec CNT100;
   1:  PR[GP1:91,1] = PR[GP1:90,1] + -55.737;
   1:  PR[GP1:91,2] = PR[GP1:90,2] + 13.636;
   1:L PR[91] R[100]mm/sec CNT100;
   1:  PR[GP1:91,1] = PR[GP1:90,1] + -57.646;
   1:  PR[GP1:91,2] = PR[GP1:90,2] + 3.105;
   1:L PR[91] R[100]mm/sec CNT100;
   1:  PR[GP1:91,1] = PR[GP1:90,1] + -58.157;
   1:  PR[GP1:91,2] = PR[GP1:90,2] + -0.066;
   1:L PR[91] R[100]mm/sec CNT100;
   1:  PR[GP1:91,1] = PR[GP1:90,1] + -56.764;
   1:  PR[GP1:91,2] = PR[GP1:90,2] + -7.721;
   1:L PR[91] R[100]mm/sec CNT100;
   1:  PR[GP1:91,1] = PR[GP1:90,1] + -56.373;
   1:  PR[GP1:91,2] = PR[GP1:90,2] + -10.331;
   1:L PR[91] R[100]mm/sec CNT100;
   1:  PR[GP1:91,1] = PR[GP1:90,1] + -55.736;
   1:  PR[GP1:91,2] = PR[GP1:90,2] + -13.782;
   1:L PR[91] R[100]mm/sec CNT100;
   1:  PR[GP1:91,1] = PR[GP1:90,1] + -50.624;
   1:  PR[GP1:91,2] = PR[GP1:90,2] + -22.429;
   1:L PR[91] R[100]mm/sec CNT100;
   1:  PR[GP1:91,1] = PR[GP1:90,1] + -48.473;
   1:  PR[GP1:91,2] = PR[GP1:90,2] + -25.988;
   1:L PR[91] R[100]mm/sec CNT100;
   1:  PR[GP1:91,1] = PR[GP1:90,1] + -41.192;
   1:  PR[GP1:91,2] = PR[GP1:90,2] + -31.994;
   1:L PR[91] R[100]mm/sec CNT100;
   1:  PR[GP1:91,1] = PR[GP1:90,1] + -37.192;
   1:  PR[GP1:91,2] = PR[GP1:90,2] + -35.160;
   1:L PR[91] R[100]mm/sec CNT100;
   1:  PR[GP1:91,1] = PR[GP1:90,1] + -29.056;
   1:  PR[GP1:91,2] = PR[GP1:90,2] + -38.159;
   1:L PR[91] R[100]mm/sec CNT100;
   1:  PR[GP1:91,1] = PR[GP1:90,1] + -23.162;
   1:  PR[GP1:91,2] = PR[GP1:90,2] + -40.092;
   1:L PR[91] R[100]mm/sec CNT100;
   1:  PR[GP1:91,1] = PR[GP1:90,1] + -15.386;
   1:  PR[GP1:91,2] = PR[GP1:90,2] + -40.231;
   1:L PR[91] R[100]mm/sec CNT100;
   1:  PR[GP1:91,1] = PR[GP1:90,1] + -8.074;
   1:  PR[GP1:91,2] = PR[GP1:90,2] + -39.970;
   1:L PR[91] R[100]mm/sec CNT100;
   1:  PR[GP1:91,1] = PR[GP1:90,1] + -1.585;
   1:  PR[GP1:91,2] = PR[GP1:90,2] + -37.954;
   1:L PR[91] R[100]mm/sec CNT100;
   1:  PR[GP1:91,1] = PR[GP1:90,1] + 1.797;
   1:  PR[GP1:91,2] = PR[GP1:90,2] + -37.953;
   1:L PR[91] R[100]mm/sec CNT100;
   1:  PR[GP1:91,1] = PR[GP1:90,1] + 8.287;
   1:  PR[GP1:91,2] = PR[GP1:90,2] + -39.969;
   1:L PR[91] R[100]mm/sec CNT100;
   1:  PR[GP1:91,1] = PR[GP1:90,1] + 15.598;
   1:  PR[GP1:91,2] = PR[GP1:90,2] + -40.230;
   1:L PR[91] R[100]mm/sec CNT100;
   1:  PR[GP1:91,1] = PR[GP1:90,1] + 23.374;
   1:  PR[GP1:91,2] = PR[GP1:90,2] + -40.093;
   1:L PR[91] R[100]mm/sec CNT100;
   1:  PR[GP1:91,1] = PR[GP1:90,1] + 29.269;
   1:  PR[GP1:91,2] = PR[GP1:90,2] + -38.159;
   1:L PR[91] R[100]mm/sec CNT100;
   1:  PR[GP1:91,1] = PR[GP1:90,1] + 37.405;
   1:  PR[GP1:91,2] = PR[GP1:90,2] + -35.162;
   1:L PR[91] R[100]mm/sec CNT100;
   1:  PR[GP1:91,1] = PR[GP1:90,1] + 41.405;
   1:  PR[GP1:91,2] = PR[GP1:90,2] + -31.995;
   1:L PR[91] R[100]mm/sec CNT100;
   1:  PR[GP1:91,1] = PR[GP1:90,1] + 48.685;
   1:  PR[GP1:91,2] = PR[GP1:90,2] + -25.983;
   1:L PR[91] R[100]mm/sec CNT100;
   1:  PR[GP1:91,1] = PR[GP1:90,1] + 50.838;
   1:  PR[GP1:91,2] = PR[GP1:90,2] + -22.425;
   1:L PR[91] R[100]mm/sec CNT100;
   1:  PR[GP1:91,1] = PR[GP1:90,1] + 55.949;
   1:  PR[GP1:91,2] = PR[GP1:90,2] + -13.797;
   1:L PR[91] R[100]mm/sec CNT100;
   1:  PR[GP1:91,1] = PR[GP1:90,1] + 57.860;
   1:  PR[GP1:91,2] = PR[GP1:90,2] + -3.249;
   1:L PR[91] R[100]mm/sec CNT100;
   1:  PR[GP1:91,1] = PR[GP1:90,1] + 58.371;
   1:  PR[GP1:91,2] = PR[GP1:90,2] + -0.078;
   1:L PR[91] R[100]mm/sec CNT100;
   1:  PR[GP1:91,1] = PR[GP1:90,1] + 56.978;
   1:  PR[GP1:91,2] = PR[GP1:90,2] + 7.586;
   1:L PR[91] R[100]mm/sec CNT100;
   1:  PR[GP1:91,1] = PR[GP1:90,1] + 56.587;
   1:  PR[GP1:91,2] = PR[GP1:90,2] + 10.198;
   1:L PR[91] R[100]mm/sec CNT100;
   1:  PR[GP1:91,1] = PR[GP1:90,1] + 55.951;
   1:  PR[GP1:91,2] = PR[GP1:90,2] + 13.650;
   1:L PR[91] R[100]mm/sec CNT100;
   1:  PR[GP1:91,1] = PR[GP1:90,1] + 50.841;
   1:  PR[GP1:91,2] = PR[GP1:90,2] + 22.277;
   1:L PR[91] R[100]mm/sec CNT100;
   1:  PR[GP1:91,1] = PR[GP1:90,1] + 48.689;
   1:  PR[GP1:91,2] = PR[GP1:90,2] + 25.835;
   1:L PR[91] R[100]mm/sec CNT100;
   1:  PR[GP1:91,1] = PR[GP1:90,1] + 41.411;
   1:  PR[GP1:91,2] = PR[GP1:90,2] + 31.848;
   1:L PR[91] R[100]mm/sec CNT100;
   1:  PR[GP1:91,1] = PR[GP1:90,1] + 37.412;
   1:  PR[GP1:91,2] = PR[GP1:90,2] + 35.014;
   1:L PR[91] R[100]mm/sec CNT100;
   1:  PR[GP1:91,1] = PR[GP1:90,1] + 29.277;
   1:  PR[GP1:91,2] = PR[GP1:90,2] + 38.014;
   1:L PR[91] R[100]mm/sec CNT100;
   1:  PR[GP1:91,1] = PR[GP1:90,1] + 23.383;
   1:  PR[GP1:91,2] = PR[GP1:90,2] + 39.947;
   1:L PR[91] R[100]mm/sec CNT100;
   1:  PR[GP1:91,1] = PR[GP1:90,1] + 15.607;
   1:  PR[GP1:91,2] = PR[GP1:90,2] + 40.088;
   1:L PR[91] R[100]mm/sec CNT100;
   1:  PR[GP1:91,1] = PR[GP1:90,1] + 8.293;
   1:  PR[GP1:91,2] = PR[GP1:90,2] + 39.826;
   1:L PR[91] R[100]mm/sec CNT100;
   1:  PR[GP1:91,1] = PR[GP1:90,1] + 1.795;
   1:  PR[GP1:91,2] = PR[GP1:90,2] + 37.822;
   1:L PR[91] R[100]mm/sec CNT100;
   1:  ! -- Layer/Ebene 140 -- !;
   1:  PR[91] = PR[90];
   1:  PR[GP1:91,1] = PR[GP1:90,1] + -1.557;
   1:  PR[GP1:91,2] = PR[GP1:90,2] + 37.996;
   1:  PR[GP1:91,3] = PR[GP1:90,3] + 85.705;
   1:L PR[91] R[100]mm/sec CNT100;
   1:  PR[GP1:91,1] = PR[GP1:90,1] + -7.783;
   1:  PR[GP1:91,2] = PR[GP1:90,2] + 39.915;
   1:L PR[91] R[100]mm/sec CNT100;
   1:  PR[GP1:91,1] = PR[GP1:90,1] + -15.433;
   1:  PR[GP1:91,2] = PR[GP1:90,2] + 40.189;
   1:L PR[91] R[100]mm/sec CNT100;
   1:  PR[GP1:91,1] = PR[GP1:90,1] + -22.909;
   1:  PR[GP1:91,2] = PR[GP1:90,2] + 40.053;
   1:L PR[91] R[100]mm/sec CNT100;
   1:  PR[GP1:91,1] = PR[GP1:90,1] + -29.134;
   1:  PR[GP1:91,2] = PR[GP1:90,2] + 38.012;
   1:L PR[91] R[100]mm/sec CNT100;
   1:  PR[GP1:91,1] = PR[GP1:90,1] + -36.977;
   1:  PR[GP1:91,2] = PR[GP1:90,2] + 35.117;
   1:L PR[91] R[100]mm/sec CNT100;
   1:  PR[GP1:91,1] = PR[GP1:90,1] + -41.259;
   1:  PR[GP1:91,2] = PR[GP1:90,2] + 31.729;
   1:L PR[91] R[100]mm/sec CNT100;
   1:  PR[GP1:91,1] = PR[GP1:90,1] + -48.292;
   1:  PR[GP1:91,2] = PR[GP1:90,2] + 25.924;
   1:L PR[91] R[100]mm/sec CNT100;
   1:  PR[GP1:91,1] = PR[GP1:90,1] + -50.635;
   1:  PR[GP1:91,2] = PR[GP1:90,2] + 22.048;
   1:L PR[91] R[100]mm/sec CNT100;
   1:  PR[GP1:91,1] = PR[GP1:90,1] + -55.579;
   1:  PR[GP1:91,2] = PR[GP1:90,2] + 13.683;
   1:L PR[91] R[100]mm/sec CNT100;
   1:  PR[GP1:91,1] = PR[GP1:90,1] + -57.426;
   1:  PR[GP1:91,2] = PR[GP1:90,2] + 3.493;
   1:L PR[91] R[100]mm/sec CNT100;
   1:  PR[GP1:91,1] = PR[GP1:90,1] + -58.000;
   1:  PR[GP1:91,2] = PR[GP1:90,2] + -0.066;
   1:L PR[91] R[100]mm/sec CNT100;
   1:  PR[GP1:91,1] = PR[GP1:90,1] + -56.715;
   1:  PR[GP1:91,2] = PR[GP1:90,2] + -7.123;
   1:L PR[91] R[100]mm/sec CNT100;
   1:  PR[GP1:91,1] = PR[GP1:90,1] + -56.283;
   1:  PR[GP1:91,2] = PR[GP1:90,2] + -10.005;
   1:L PR[91] R[100]mm/sec CNT100;
   1:  PR[GP1:91,1] = PR[GP1:90,1] + -55.578;
   1:  PR[GP1:91,2] = PR[GP1:90,2] + -13.829;
   1:L PR[91] R[100]mm/sec CNT100;
   1:  PR[GP1:91,1] = PR[GP1:90,1] + -50.631;
   1:  PR[GP1:91,2] = PR[GP1:90,2] + -22.196;
   1:L PR[91] R[100]mm/sec CNT100;
   1:  PR[GP1:91,1] = PR[GP1:90,1] + -48.288;
   1:  PR[GP1:91,2] = PR[GP1:90,2] + -26.072;
   1:L PR[91] R[100]mm/sec CNT100;
   1:  PR[GP1:91,1] = PR[GP1:90,1] + -41.252;
   1:  PR[GP1:91,2] = PR[GP1:90,2] + -31.876;
   1:L PR[91] R[100]mm/sec CNT100;
   1:  PR[GP1:91,1] = PR[GP1:90,1] + -36.971;
   1:  PR[GP1:91,2] = PR[GP1:90,2] + -35.265;
   1:L PR[91] R[100]mm/sec CNT100;
   1:  PR[GP1:91,1] = PR[GP1:90,1] + -29.125;
   1:  PR[GP1:91,2] = PR[GP1:90,2] + -38.157;
   1:L PR[91] R[100]mm/sec CNT100;
   1:  PR[GP1:91,1] = PR[GP1:90,1] + -22.901;
   1:  PR[GP1:91,2] = PR[GP1:90,2] + -40.198;
   1:L PR[91] R[100]mm/sec CNT100;
   1:  PR[GP1:91,1] = PR[GP1:90,1] + -15.424;
   1:  PR[GP1:91,2] = PR[GP1:90,2] + -40.331;
   1:L PR[91] R[100]mm/sec CNT100;
   1:  PR[GP1:91,1] = PR[GP1:90,1] + -7.777;
   1:  PR[GP1:91,2] = PR[GP1:90,2] + -40.059;
   1:L PR[91] R[100]mm/sec CNT100;
   1:  PR[GP1:91,1] = PR[GP1:90,1] + -1.559;
   1:  PR[GP1:91,2] = PR[GP1:90,2] + -38.128;
   1:L PR[91] R[100]mm/sec CNT100;
   1:  PR[GP1:91,1] = PR[GP1:90,1] + 1.772;
   1:  PR[GP1:91,2] = PR[GP1:90,2] + -38.127;
   1:L PR[91] R[100]mm/sec CNT100;
   1:  PR[GP1:91,1] = PR[GP1:90,1] + 7.990;
   1:  PR[GP1:91,2] = PR[GP1:90,2] + -40.058;
   1:L PR[91] R[100]mm/sec CNT100;
   1:  PR[GP1:91,1] = PR[GP1:90,1] + 15.637;
   1:  PR[GP1:91,2] = PR[GP1:90,2] + -40.331;
   1:L PR[91] R[100]mm/sec CNT100;
   1:  PR[GP1:91,1] = PR[GP1:90,1] + 23.114;
   1:  PR[GP1:91,2] = PR[GP1:90,2] + -40.199;
   1:L PR[91] R[100]mm/sec CNT100;
   1:  PR[GP1:91,1] = PR[GP1:90,1] + 29.338;
   1:  PR[GP1:91,2] = PR[GP1:90,2] + -38.157;
   1:L PR[91] R[100]mm/sec CNT100;
   1:  PR[GP1:91,1] = PR[GP1:90,1] + 37.184;
   1:  PR[GP1:91,2] = PR[GP1:90,2] + -35.267;
   1:L PR[91] R[100]mm/sec CNT100;
   1:  PR[GP1:91,1] = PR[GP1:90,1] + 41.465;
   1:  PR[GP1:91,2] = PR[GP1:90,2] + -31.877;
   1:L PR[91] R[100]mm/sec CNT100;
   1:  PR[GP1:91,1] = PR[GP1:90,1] + 48.501;
   1:  PR[GP1:91,2] = PR[GP1:90,2] + -26.067;
   1:L PR[91] R[100]mm/sec CNT100;
   1:  PR[GP1:91,1] = PR[GP1:90,1] + 50.845;
   1:  PR[GP1:91,2] = PR[GP1:90,2] + -22.193;
   1:L PR[91] R[100]mm/sec CNT100;
   1:  PR[GP1:91,1] = PR[GP1:90,1] + 55.791;
   1:  PR[GP1:91,2] = PR[GP1:90,2] + -13.844;
   1:L PR[91] R[100]mm/sec CNT100;
   1:  PR[GP1:91,1] = PR[GP1:90,1] + 57.639;
   1:  PR[GP1:91,2] = PR[GP1:90,2] + -3.638;
   1:L PR[91] R[100]mm/sec CNT100;
   1:  PR[GP1:91,1] = PR[GP1:90,1] + 58.213;
   1:  PR[GP1:91,2] = PR[GP1:90,2] + -0.078;
   1:L PR[91] R[100]mm/sec CNT100;
   1:  PR[GP1:91,1] = PR[GP1:90,1] + 56.929;
   1:  PR[GP1:91,2] = PR[GP1:90,2] + 6.987;
   1:L PR[91] R[100]mm/sec CNT100;
   1:  PR[GP1:91,1] = PR[GP1:90,1] + 56.498;
   1:  PR[GP1:91,2] = PR[GP1:90,2] + 9.872;
   1:L PR[91] R[100]mm/sec CNT100;
   1:  PR[GP1:91,1] = PR[GP1:90,1] + 55.792;
   1:  PR[GP1:91,2] = PR[GP1:90,2] + 13.697;
   1:L PR[91] R[100]mm/sec CNT100;
   1:  PR[GP1:91,1] = PR[GP1:90,1] + 50.848;
   1:  PR[GP1:91,2] = PR[GP1:90,2] + 22.045;
   1:L PR[91] R[100]mm/sec CNT100;
   1:  PR[GP1:91,1] = PR[GP1:90,1] + 48.505;
   1:  PR[GP1:91,2] = PR[GP1:90,2] + 25.919;
   1:L PR[91] R[100]mm/sec CNT100;
   1:  PR[GP1:91,1] = PR[GP1:90,1] + 41.471;
   1:  PR[GP1:91,2] = PR[GP1:90,2] + 31.730;
   1:L PR[91] R[100]mm/sec CNT100;
   1:  PR[GP1:91,1] = PR[GP1:90,1] + 37.190;
   1:  PR[GP1:91,2] = PR[GP1:90,2] + 35.119;
   1:L PR[91] R[100]mm/sec CNT100;
   1:  PR[GP1:91,1] = PR[GP1:90,1] + 29.346;
   1:  PR[GP1:91,2] = PR[GP1:90,2] + 38.012;
   1:L PR[91] R[100]mm/sec CNT100;
   1:  PR[GP1:91,1] = PR[GP1:90,1] + 23.122;
   1:  PR[GP1:91,2] = PR[GP1:90,2] + 40.053;
   1:L PR[91] R[100]mm/sec CNT100;
   1:  PR[GP1:91,1] = PR[GP1:90,1] + 15.646;
   1:  PR[GP1:91,2] = PR[GP1:90,2] + 40.189;
   1:L PR[91] R[100]mm/sec CNT100;
   1:  PR[GP1:91,1] = PR[GP1:90,1] + 7.996;
   1:  PR[GP1:91,2] = PR[GP1:90,2] + 39.915;
   1:L PR[91] R[100]mm/sec CNT100;
   1:  PR[GP1:91,1] = PR[GP1:90,1] + 1.770;
   1:  PR[GP1:91,2] = PR[GP1:90,2] + 37.995;
   1:L PR[91] R[100]mm/sec CNT100;
   1:  ! -- Layer/Ebene 141 -- !;
   1:  PR[91] = PR[90];
   1:  PR[GP1:91,1] = PR[GP1:90,1] + -1.532;
   1:  PR[GP1:91,2] = PR[GP1:90,2] + 38.169;
   1:  PR[GP1:91,3] = PR[GP1:90,3] + 86.315;
   1:L PR[91] R[100]mm/sec CNT100;
   1:  PR[GP1:91,1] = PR[GP1:90,1] + -7.485;
   1:  PR[GP1:91,2] = PR[GP1:90,2] + 40.004;
   1:L PR[91] R[100]mm/sec CNT100;
   1:  PR[GP1:91,1] = PR[GP1:90,1] + -15.471;
   1:  PR[GP1:91,2] = PR[GP1:90,2] + 40.290;
   1:L PR[91] R[100]mm/sec CNT100;
   1:  PR[GP1:91,1] = PR[GP1:90,1] + -22.648;
   1:  PR[GP1:91,2] = PR[GP1:90,2] + 40.159;
   1:L PR[91] R[100]mm/sec CNT100;
   1:  PR[GP1:91,1] = PR[GP1:90,1] + -29.202;
   1:  PR[GP1:91,2] = PR[GP1:90,2] + 38.010;
   1:L PR[91] R[100]mm/sec CNT100;
   1:  PR[GP1:91,1] = PR[GP1:90,1] + -36.756;
   1:  PR[GP1:91,2] = PR[GP1:90,2] + 35.222;
   1:L PR[91] R[100]mm/sec CNT100;
   1:  PR[GP1:91,1] = PR[GP1:90,1] + -41.319;
   1:  PR[GP1:91,2] = PR[GP1:90,2] + 31.611;
   1:L PR[91] R[100]mm/sec CNT100;
   1:  PR[GP1:91,1] = PR[GP1:90,1] + -48.107;
   1:  PR[GP1:91,2] = PR[GP1:90,2] + 26.008;
   1:L PR[91] R[100]mm/sec CNT100;
   1:  PR[GP1:91,1] = PR[GP1:90,1] + -50.642;
   1:  PR[GP1:91,2] = PR[GP1:90,2] + 21.815;
   1:L PR[91] R[100]mm/sec CNT100;
   1:  PR[GP1:91,1] = PR[GP1:90,1] + -55.420;
   1:  PR[GP1:91,2] = PR[GP1:90,2] + 13.730;
   1:L PR[91] R[100]mm/sec CNT100;
   1:  PR[GP1:91,1] = PR[GP1:90,1] + -57.206;
   1:  PR[GP1:91,2] = PR[GP1:90,2] + 3.881;
   1:L PR[91] R[100]mm/sec CNT100;
   1:  PR[GP1:91,1] = PR[GP1:90,1] + -57.842;
   1:  PR[GP1:91,2] = PR[GP1:90,2] + -0.066;
   1:L PR[91] R[100]mm/sec CNT100;
   1:  PR[GP1:91,1] = PR[GP1:90,1] + -56.666;
   1:  PR[GP1:91,2] = PR[GP1:90,2] + -6.525;
   1:L PR[91] R[100]mm/sec CNT100;
   1:  PR[GP1:91,1] = PR[GP1:90,1] + -56.194;
   1:  PR[GP1:91,2] = PR[GP1:90,2] + -9.680;
   1:L PR[91] R[100]mm/sec CNT100;
   1:  PR[GP1:91,1] = PR[GP1:90,1] + -55.420;
   1:  PR[GP1:91,2] = PR[GP1:90,2] + -13.876;
   1:L PR[91] R[100]mm/sec CNT100;
   1:  PR[GP1:91,1] = PR[GP1:90,1] + -50.639;
   1:  PR[GP1:91,2] = PR[GP1:90,2] + -21.963;
   1:L PR[91] R[100]mm/sec CNT100;
   1:  PR[GP1:91,1] = PR[GP1:90,1] + -48.104;
   1:  PR[GP1:91,2] = PR[GP1:90,2] + -26.156;
   1:L PR[91] R[100]mm/sec CNT100;
   1:  PR[GP1:91,1] = PR[GP1:90,1] + -41.312;
   1:  PR[GP1:91,2] = PR[GP1:90,2] + -31.758;
   1:L PR[91] R[100]mm/sec CNT100;
   1:  PR[GP1:91,1] = PR[GP1:90,1] + -36.750;
   1:  PR[GP1:91,2] = PR[GP1:90,2] + -35.369;
   1:L PR[91] R[100]mm/sec CNT100;
   1:  PR[GP1:91,1] = PR[GP1:90,1] + -29.194;
   1:  PR[GP1:91,2] = PR[GP1:90,2] + -38.154;
   1:L PR[91] R[100]mm/sec CNT100;
   1:  PR[GP1:91,1] = PR[GP1:90,1] + -22.640;
   1:  PR[GP1:91,2] = PR[GP1:90,2] + -40.305;
   1:L PR[91] R[100]mm/sec CNT100;
   1:  PR[GP1:91,1] = PR[GP1:90,1] + -15.463;
   1:  PR[GP1:91,2] = PR[GP1:90,2] + -40.432;
   1:L PR[91] R[100]mm/sec CNT100;
   1:  PR[GP1:91,1] = PR[GP1:90,1] + -7.480;
   1:  PR[GP1:91,2] = PR[GP1:90,2] + -40.147;
   1:L PR[91] R[100]mm/sec CNT100;
   1:  PR[GP1:91,1] = PR[GP1:90,1] + -1.534;
   1:  PR[GP1:91,2] = PR[GP1:90,2] + -38.301;
   1:L PR[91] R[100]mm/sec CNT100;
   1:  PR[GP1:91,1] = PR[GP1:90,1] + 1.747;
   1:  PR[GP1:91,2] = PR[GP1:90,2] + -38.300;
   1:L PR[91] R[100]mm/sec CNT100;
   1:  PR[GP1:91,1] = PR[GP1:90,1] + 7.693;
   1:  PR[GP1:91,2] = PR[GP1:90,2] + -40.147;
   1:L PR[91] R[100]mm/sec CNT100;
   1:  PR[GP1:91,1] = PR[GP1:90,1] + 15.676;
   1:  PR[GP1:91,2] = PR[GP1:90,2] + -40.431;
   1:L PR[91] R[100]mm/sec CNT100;
   1:  PR[GP1:91,1] = PR[GP1:90,1] + 22.853;
   1:  PR[GP1:91,2] = PR[GP1:90,2] + -40.305;
   1:L PR[91] R[100]mm/sec CNT100;
   1:  PR[GP1:91,1] = PR[GP1:90,1] + 29.406;
   1:  PR[GP1:91,2] = PR[GP1:90,2] + -38.155;
   1:L PR[91] R[100]mm/sec CNT100;
   1:  PR[GP1:91,1] = PR[GP1:90,1] + 36.963;
   1:  PR[GP1:91,2] = PR[GP1:90,2] + -35.371;
   1:L PR[91] R[100]mm/sec CNT100;
   1:  PR[GP1:91,1] = PR[GP1:90,1] + 41.525;
   1:  PR[GP1:91,2] = PR[GP1:90,2] + -31.759;
   1:L PR[91] R[100]mm/sec CNT100;
   1:  PR[GP1:91,1] = PR[GP1:90,1] + 48.317;
   1:  PR[GP1:91,2] = PR[GP1:90,2] + -26.151;
   1:L PR[91] R[100]mm/sec CNT100;
   1:  PR[GP1:91,1] = PR[GP1:90,1] + 50.852;
   1:  PR[GP1:91,2] = PR[GP1:90,2] + -21.960;
   1:L PR[91] R[100]mm/sec CNT100;
   1:  PR[GP1:91,1] = PR[GP1:90,1] + 55.632;
   1:  PR[GP1:91,2] = PR[GP1:90,2] + -13.891;
   1:L PR[91] R[100]mm/sec CNT100;
   1:  PR[GP1:91,1] = PR[GP1:90,1] + 57.419;
   1:  PR[GP1:91,2] = PR[GP1:90,2] + -4.026;
   1:L PR[91] R[100]mm/sec CNT100;
   1:  PR[GP1:91,1] = PR[GP1:90,1] + 58.055;
   1:  PR[GP1:91,2] = PR[GP1:90,2] + -0.078;
   1:L PR[91] R[100]mm/sec CNT100;
   1:  PR[GP1:91,1] = PR[GP1:90,1] + 56.880;
   1:  PR[GP1:91,2] = PR[GP1:90,2] + 6.388;
   1:L PR[91] R[100]mm/sec CNT100;
   1:  PR[GP1:91,1] = PR[GP1:90,1] + 56.408;
   1:  PR[GP1:91,2] = PR[GP1:90,2] + 9.546;
   1:L PR[91] R[100]mm/sec CNT100;
   1:  PR[GP1:91,1] = PR[GP1:90,1] + 55.634;
   1:  PR[GP1:91,2] = PR[GP1:90,2] + 13.744;
   1:L PR[91] R[100]mm/sec CNT100;
   1:  PR[GP1:91,1] = PR[GP1:90,1] + 50.855;
   1:  PR[GP1:91,2] = PR[GP1:90,2] + 21.812;
   1:L PR[91] R[100]mm/sec CNT100;
   1:  PR[GP1:91,1] = PR[GP1:90,1] + 48.320;
   1:  PR[GP1:91,2] = PR[GP1:90,2] + 26.003;
   1:L PR[91] R[100]mm/sec CNT100;
   1:  PR[GP1:91,1] = PR[GP1:90,1] + 41.531;
   1:  PR[GP1:91,2] = PR[GP1:90,2] + 31.612;
   1:L PR[91] R[100]mm/sec CNT100;
   1:  PR[GP1:91,1] = PR[GP1:90,1] + 36.969;
   1:  PR[GP1:91,2] = PR[GP1:90,2] + 35.224;
   1:L PR[91] R[100]mm/sec CNT100;
   1:  PR[GP1:91,1] = PR[GP1:90,1] + 29.415;
   1:  PR[GP1:91,2] = PR[GP1:90,2] + 38.010;
   1:L PR[91] R[100]mm/sec CNT100;
   1:  PR[GP1:91,1] = PR[GP1:90,1] + 22.861;
   1:  PR[GP1:91,2] = PR[GP1:90,2] + 40.159;
   1:L PR[91] R[100]mm/sec CNT100;
   1:  PR[GP1:91,1] = PR[GP1:90,1] + 15.684;
   1:  PR[GP1:91,2] = PR[GP1:90,2] + 40.289;
   1:L PR[91] R[100]mm/sec CNT100;
   1:  PR[GP1:91,1] = PR[GP1:90,1] + 7.698;
   1:  PR[GP1:91,2] = PR[GP1:90,2] + 40.003;
   1:L PR[91] R[100]mm/sec CNT100;
   1:  PR[GP1:91,1] = PR[GP1:90,1] + 1.745;
   1:  PR[GP1:91,2] = PR[GP1:90,2] + 38.169;
   1:L PR[91] R[100]mm/sec CNT100 TB   .50sec,CALL END_PUD;
   1:  DO[117:Laser Start]=OFF;
   1:  !Sicherheitspunkt!;
   1:  PR[92] = PR[91];
   1:  PR[92] = PR[GP1:92,3] + 50;
   1:J PR[92];
   1:  WAIT   5.00(sec);
   1:  DO[119:Gas]=OFF;
   1:  CALL HOME_ALL;
/POS
/END
